KUKA KRL program: MyProgram_050().src

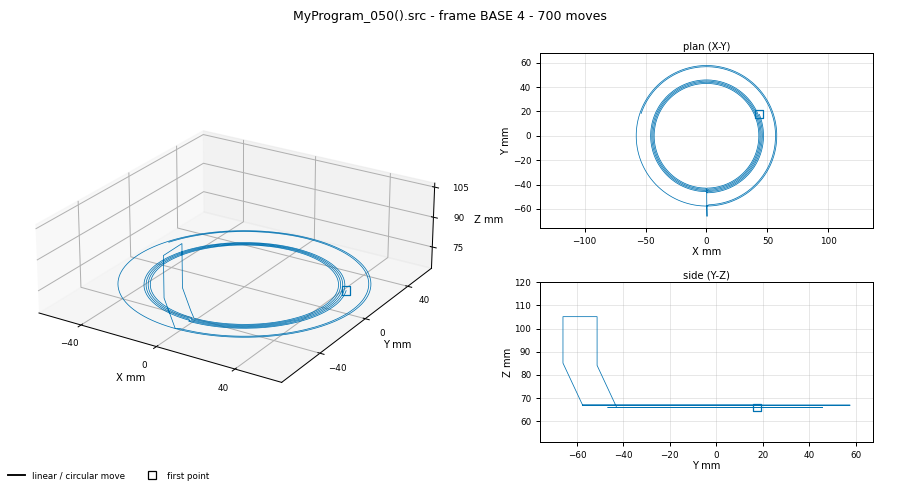
[picture p0: tool path of MyProgram_050().src in frame BASE 4, 700 of 700 moves have a stored position in this frame; points joined in program order, loops and branches not executed]
&ACCESS RVP
&REL 1
&PARAM TEMPLATE = C:\KRC\Roboter\Template\vorgabe
&PARAM EDITMASK = *
DEF MyProgram_050()
; ---- Setting reference (Base) ----
$BASE = BASE_DATA[4]

; --------------------------
; ---- Setting tool (TCP) ----
$TOOL = TOOL_DATA[3]
; --------------------------

$VEL.CP = VEL_APROX_PRINT
Startdeposition()
$VEL.CP = VEL_PRINT
LIN {X 43.3349,Y 17.5684,Z 66,A 14.5783,B 24.8507,C -2.8194,E1 25.1489,E2 68.8422} C_DIS
LIN {X 44.2203,Y 15.2025,Z 66,A 11.1131,B 24.8523,C -2.8036,E1 25.1522,E2 72.3254} C_DIS
LIN {X 45.3904,Y 11.2372,Z 66,A 5.962,B 24.8541,C -2.7869,E1 25.156,E2 77.4863} C_DIS
LIN {X 46.2102,Y 7.1538,Z 66,A 1.4001,B 24.8547,C -2.7815,E1 25.1582,E2 82.0343} C_DIS
LIN {X 46.518,Y 4.7576,Z 66,A -1.6458,B 24.8558,C -2.7707,E1 25.1592,E2 85.0877} C_DIS
LIN {X 46.6896,Y 2.5751,Z 66,A -4.0137,B 24.8561,C -2.7683,E1 25.1596,E2 87.4473} C_DIS
LIN {X 46.7545,Y 0.7633,Z 66,A -6.5593,B 24.8574,C -2.7552,E1 25.1598,E2 90.0088} C_DIS
LIN {X 46.695,Y -2.4713,Z 66,A -10.1755,B 24.858,C -2.7493,E1 25.1595,E2 93.6174} C_DIS
LIN {X 46.5699,Y -4.2183,Z 66,A -12.454,B 24.859,C -2.74,E1 25.1589,E2 95.9043} C_DIS
LIN {X 46.2757,Y -6.7166,Z 66,A -15.3552,B 24.8596,C -2.7338,E1 25.1579,E2 98.8032} C_DIS
LIN {X 45.8823,Y -9.0213,Z 66,A -18.6554,B 24.8614,C -2.7165,E1 25.1562,E2 102.1248} C_DIS
LIN {X 45.206,Y -11.9579,Z 66,A -22.2433,B 24.8624,C -2.7071,E1 25.1538,E2 105.7144} C_DIS
LIN {X 44.3153,Y -14.9224,Z 66,A -25.7557,B 24.863,C -2.7008,E1 25.1508,E2 109.2217} C_DIS
LIN {X 43.3729,Y -17.4745,Z 66,A -29.1739,B 24.8642,C -2.6891,E1 25.1474,E2 112.6486} C_DIS
LIN {X 42.3193,Y -19.8908,Z 66,A -32.2612,B 24.8649,C -2.6822,E1 25.1438,E2 115.7353} C_DIS
LIN {X 40.7412,Y -22.9499,Z 66,A -37.2752,B 24.8676,C -2.6553,E1 25.1371,E2 120.7867} C_DIS
LIN {X 38.8256,Y -26.0596,Z 66,A -41.3629,B 24.8681,C -2.6501,E1 25.1309,E2 124.8663} C_DIS
LIN {X 36.3077,Y -29.4671,Z 66,A -46.4536,B 24.8693,C -2.6384,E1 25.1222,E2 129.9607} C_DIS
LIN {X 34.1441,Y -31.9491,Z 66,A -49.9088,B 24.8693,C -2.6389,E1 25.1158,E2 133.3991} C_DIS
LIN {X 32.775,Y -33.3522,Z 66,A -52.3553,B 24.8699,C -2.6324,E1 25.111,E2 135.8507} C_DIS
LIN {X 31.3542,Y -34.6908,Z 66,A -54.822,B 24.8706,C -2.6255,E1 25.1059,E2 138.3236} C_DIS
LIN {X 29.1349,Y -36.5752,Z 66,A -59.1688,B 24.8727,C -2.6038,E1 25.0964,E2 142.7054} C_DIS
LIN {X 25.3481,Y -39.2942,Z 66,A -63.9176,B 24.8721,C -2.6097,E1 25.0856,E2 147.424} C_DIS
LIN {X 22.2733,Y -41.1151,Z 66,A -69.1086,B 24.8743,C -2.5878,E1 25.0729,E2 152.6516} C_DIS
LIN {X 19.1514,Y -42.6589,Z 66,A -72.7416,B 24.8738,C -2.5922,E1 25.0638,E2 156.2648} C_DIS
LIN {X 16.7047,Y -43.6749,Z 66,A -76.1469,B 24.8745,C -2.585,E1 25.0549,E2 159.6795} C_DIS
LIN {X 14.3201,Y -44.5136,Z 66,A -79.3958,B 24.8752,C -2.5787,E1 25.0463,E2 162.9371} C_DIS
LIN {X 11.2683,Y -45.3827,Z 66,A -82.4317,B 24.8742,C -2.589,E1 25.0382,E2 165.9436} C_DIS
LIN {X 9.0342,Y -45.8799,Z 66,A -86.2122,B 24.876,C -2.5702,E1 25.0277,E2 169.7639} C_DIS
LIN {X 6.7643,Y -46.269,Z 66,A -88.946,B 24.876,C -2.5697,E1 25.0202,E2 172.4964} C_DIS
LIN {X 2.9921,Y -46.665,Z 66,A -93.1614,B 24.8756,C -2.5744,E1 25.0085,E2 176.6981} C_DIS
LIN {X 0.2144,Y -46.7557,Z 66,A -95.0475,B 24.8733,C -2.5983,E1 25.0034,E2 178.5272} C_DIS
Enddeposition()
LIN {X 0.2144,Y -46.7557,Z 66,A -95.0475,B 24.8733,C -2.5983,E1 25.0034,E2 178.5272} C_DIS
Startdeposition()
$VEL.CP = VEL_PRINT
LIN {X 0.8978,Y -45.7928,Z 66,A -94.2069,B 24.8717,C -2.6146,E1 25.0059,E2 177.648} C_DIS
LIN {X 2.9762,Y -45.7048,Z 66,A -91.241,B 24.871,C -2.6216,E1 25.0142,E2 174.6666} C_DIS
LIN {X 6.5228,Y -45.3347,Z 66,A -87.6101,B 24.872,C -2.6106,E1 25.0242,E2 171.0646} C_DIS
LIN {X 7.8991,Y -45.1153,Z 66,A -85.4528,B 24.8712,C -2.6188,E1 25.0301,E2 168.8902} C_DIS
LIN {X 10.8381,Y -44.5008,Z 66,A -81.704,B 24.8709,C -2.6221,E1 25.0404,E2 165.1385} C_DIS
LIN {X 13.368,Y -43.8073,Z 66,A -78.1682,B 24.8701,C -2.63,E1 25.0499,E2 161.5899} C_DIS
LIN {X 15.9038,Y -42.9513,Z 66,A -75.1389,B 24.8702,C -2.6288,E1 25.0578,E2 158.5697} C_DIS
LIN {X 18.2204,Y -42.0213,Z 66,A -72.3421,B 24.8704,C -2.6275,E1 25.065,E2 155.7823} C_DIS
LIN {X 19.5156,Y -41.436,Z 66,A -69.8624,B 24.8689,C -2.6425,E1 25.0714,E2 153.2734} C_DIS
LIN {X 22.8629,Y -39.6867,Z 66,A -65.528,B 24.8688,C -2.6437,E1 25.082,E2 148.9489} C_DIS
LIN {X 24.7649,Y -38.529,Z 66,A -62.1736,B 24.8672,C -2.6591,E1 25.0899,E2 145.5687} C_DIS
LIN {X 28.2935,Y -36.0177,Z 66,A -57.8091,B 24.868,C -2.6512,E1 25.0997,E2 141.2385} C_DIS
LIN {X 30.3014,Y -34.346,Z 66,A -53.7652,B 24.8659,C -2.6725,E1 25.1083,E2 137.16} C_DIS
LIN {X 32.0835,Y -32.6872,Z 66,A -51.4223,B 24.8665,C -2.6667,E1 25.113,E2 134.8403} C_DIS
LIN {X 34.0299,Y -30.6556,Z 66,A -47.0128,B 24.8639,C -2.6918,E1 25.1214,E2 130.3909} C_DIS
LIN {X 35.7191,Y -28.6702,Z 66,A -43.7714,B 24.8631,C -2.6998,E1 25.1271,E2 127.1455} C_DIS
LIN {X 38.0986,Y -25.4232,Z 66,A -39.7855,B 24.8637,C -2.6938,E1 25.1335,E2 123.1933} C_DIS
LIN {X 39.2143,Y -23.6641,Z 66,A -36.3538,B 24.8614,C -2.7165,E1 25.1386,E2 119.7252} C_DIS
LIN {X 41.065,Y -20.2842,Z 66,A -32.2707,B 24.8614,C -2.7165,E1 25.1439,E2 115.6637} C_DIS
LIN {X 41.7032,Y -18.9371,Z 66,A -30.0884,B 24.8602,C -2.728,E1 25.1465,E2 113.466} C_DIS
LIN {X 42.7319,Y -16.4845,Z 66,A -27.0475,B 24.8598,C -2.7326,E1 25.1497,E2 110.4311} C_DIS
LIN {X 43.2185,Y -15.1634,Z 66,A -24.779,B 24.8582,C -2.7475,E1 25.1518,E2 108.1399} C_DIS
LIN {X 44.2475,Y -11.8303,Z 66,A -20.9893,B 24.858,C -2.75,E1 25.1547,E2 104.3659} C_DIS
LIN {X 44.7342,Y -9.8304,Z 66,A -18.011,B 24.8563,C -2.7657,E1 25.1566,E2 101.3678} C_DIS
LIN {X 45.1853,Y -7.488,Z 66,A -14.8477,B 24.855,C -2.7785,E1 25.1581,E2 98.1929} C_DIS
LIN {X 45.6688,Y -3.4865,Z 66,A -10.5749,B 24.8549,C -2.7797,E1 25.1594,E2 93.9426} C_DIS
LIN {X 45.7926,Y -0.9082,Z 66,A -6.6136,B 24.8523,C -2.8038,E1 25.1598,E2 89.9477} C_DIS
LIN {X 45.7713,Y 1.6691,Z 66,A -3.6991,B 24.8519,C -2.808,E1 25.1596,E2 87.0407} C_DIS
LIN {X 45.5857,Y 4.4425,Z 66,A -0.6525,B 24.8516,C -2.8107,E1 25.1589,E2 84.0058} C_DIS
LIN {X 45.3638,Y 6.3188,Z 66,A 1.9954,B 24.8503,C -2.8233,E1 25.1579,E2 81.3435} C_DIS
LIN {X 45.0043,Y 8.508,Z 66,A 4.7588,B 24.8494,C -2.8316,E1 25.1566,E2 78.5769} C_DIS
LIN {X 44.4208,Y 11.161,Z 66,A 7.5921,B 24.8494,C -2.8312,E1 25.1548,E2 75.7609} C_DIS
LIN {X 43.4383,Y 14.5227,Z 66,A 12.5584,B 24.8469,C -2.8551,E1 25.1508,E2 70.7665} C_DIS
LIN {X 42.4975,Y 17.0812,Z 66,A 15.8627,B 24.846,C -2.8628,E1 25.1475,E2 67.4622} C_DIS
LIN {X 41.091,Y 20.2317,Z 66,A 20.3435,B 24.8444,C -2.8778,E1 25.1422,E2 62.9701} C_DIS
LIN {X 39.4422,Y 23.283,Z 66,A 24.8067,B 24.8429,C -2.8915,E1 25.1361,E2 58.4976} C_DIS
LIN {X 37.4354,Y 26.3899,Z 66,A 29.3094,B 24.8419,C -2.9007,E1 25.129,E2 53.9953} C_DIS
LIN {X 35.8889,Y 28.4565,Z 66,A 32.3347,B 24.8415,C -2.9047,E1 25.1239,E2 50.9751} C_DIS
LIN {X 33.9496,Y 30.7449,Z 66,A 35.9504,B 24.8408,C -2.9106,E1 25.1173,E2 47.3616} C_DIS
LIN {X 32.4039,Y 32.37,Z 66,A 38.5786,B 24.8405,C -2.9133,E1 25.1122,E2 44.7381} C_DIS
LIN {X 30.8201,Y 33.8814,Z 66,A 41.5735,B 24.8394,C -2.9233,E1 25.106,E2 41.7318} C_DIS
LIN {X 28.9064,Y 35.5276,Z 66,A 44.755,B 24.8387,C -2.9296,E1 25.0992,E2 38.5476} C_DIS
LIN {X 26.0164,Y 37.6956,Z 66,A 48.8498,B 24.8387,C -2.9299,E1 25.09,E2 34.4667} C_DIS
LIN {X 23.2214,Y 39.4786,Z 66,A 52.9902,B 24.838,C -2.936,E1 25.0802,E2 30.3251} C_DIS
LIN {X 20.8606,Y 40.7752,Z 66,A 56.8481,B 24.8366,C -2.9487,E1 25.0707,E2 26.448} C_DIS
LIN {X 18.7515,Y 41.7872,Z 66,A 60.2609,B 24.8353,C -2.9602,E1 25.0619,E2 23.0165} C_DIS
LIN {X 16.1644,Y 42.8544,Z 66,A 62.9926,B 24.8364,C -2.9507,E1 25.0549,E2 20.3134} C_DIS
LIN {X 13.9943,Y 43.6114,Z 66,A 65.9425,B 24.836,C -2.9542,E1 25.0471,E2 17.3607} C_DIS
LIN {X 11.6913,Y 44.2844,Z 66,A 69.7433,B 24.8343,C -2.9692,E1 25.0368,E2 13.5304} C_DIS
LIN {X 8.6249,Y 44.9822,Z 66,A 73.6023,B 24.8343,C -2.9697,E1 25.0262,E2 9.6749} C_DIS
LIN {X 3.9155,Y 45.634,Z 66,A 78.5134,B 24.836,C -2.9542,E1 25.0127,E2 4.8043} C_DIS
LIN {X 1.0821,Y 45.7888,Z 66,A 82.7236,B 24.8349,C -2.9643,E1 25.0009,E2 0.5713} C_DIS
LIN {X -1.5721,Y 45.7747,Z 66,A 85.9582,B 24.8351,C -2.9621,E1 24.9919,E2 -2.6583} C_DIS
LIN {X -4.9742,Y 45.5306,Z 66,A 90.0108,B 24.8357,C -2.9568,E1 24.9806,E2 -6.7003} C_DIS
LIN {X -7.4603,Y 45.19,Z 66,A 93.4271,B 24.8355,C -2.9589,E1 24.9712,E2 -10.1245} C_DIS
LIN {X -9.7479,Y 44.7522,Z 66,A 96.3601,B 24.8357,C -2.9567,E1 24.9632,E2 -13.056} C_DIS
LIN {X -13.1885,Y 43.8617,Z 66,A 100.5053,B 24.8367,C -2.9478,E1 24.9521,E2 -17.1862} C_DIS
LIN {X -16.3693,Y 42.7765,Z 66,A 104.5263,B 24.8376,C -2.94,E1 24.9415,E2 -21.1966} C_DIS
LIN {X -18.0147,Y 42.1101,Z 66,A 106.8564,B 24.8377,C -2.9384,E1 24.9355,E2 -23.5283} C_DIS
LIN {X -20.0814,Y 41.1647,Z 66,A 109.6892,B 24.8382,C -2.934,E1 24.9284,E2 -26.3577} C_DIS
LIN {X -22.1767,Y 40.075,Z 66,A 113.1651,B 24.838,C -2.9364,E1 24.9198,E2 -29.849} C_DIS
LIN {X -24.6187,Y 38.6228,Z 66,A 116.1352,B 24.8396,C -2.9218,E1 24.9128,E2 -32.7938} C_DIS
LIN {X -26.8632,Y 37.097,Z 66,A 120.1797,B 24.8393,C -2.9241,E1 24.9035,E2 -36.8574} C_DIS
LIN {X -29.4193,Y 35.1045,Z 66,A 123.6418,B 24.8412,C -2.9075,E1 24.896,E2 -40.2928} C_DIS
LIN {X -30.6738,Y 34.0124,Z 66,A 126.2288,B 24.8409,C -2.9096,E1 24.8906,E2 -42.8952} C_DIS
LIN {X -33.081,Y 31.6774,Z 66,A 130.4532,B 24.842,C -2.9,E1 24.8823,E2 -47.1148} C_DIS
LIN {X -35.5132,Y 28.9239,Z 66,A 134.4029,B 24.8442,C -2.8801,E1 24.8752,E2 -51.0347} C_DIS
LIN {X -36.3677,Y 27.8421,Z 66,A 136.3444,B 24.8443,C -2.8784,E1 24.8719,E2 -52.9813} C_DIS
LIN {X -37.8873,Y 25.736,Z 66,A 140.0753,B 24.8446,C -2.8759,E1 24.8659,E2 -56.7246} C_DIS
LIN {X -39.2931,Y 23.5348,Z 66,A 143.5261,B 24.8453,C -2.8692,E1 24.8609,E2 -60.1771} C_DIS
LIN {X -41.2526,Y 19.9,Z 66,A 148.3302,B 24.8474,C -2.8497,E1 24.8547,E2 -64.9601} C_DIS
LIN {X -42.3378,Y 17.4725,Z 66,A 151.8219,B 24.8483,C -2.8419,E1 24.8509,E2 -68.4526} C_DIS
LIN {X -43.324,Y 14.8597,Z 66,A 155.0988,B 24.8497,C -2.8286,E1 24.8478,E2 -71.7163} C_DIS
LIN {X -43.9589,Y 12.861,Z 66,A 157.5559,B 24.8508,C -2.8185,E1 24.8458,E2 -74.1634} C_DIS
LIN {X -44.6534,Y 10.1894,Z 66,A 161.8476,B 24.8508,C -2.8184,E1 24.843,E2 -78.4799} C_DIS
LIN {X -45.4195,Y 5.9038,Z 66,A 166.3561,B 24.8538,C -2.7895,E1 24.841,E2 -82.9462} C_DIS
LIN {X -45.626,Y 4.0058,Z 66,A 169.1778,B 24.8541,C -2.7874,E1 24.8402,E2 -85.7797} C_DIS
LIN {X -45.7994,Y 0.4243,Z 66,A 173.4393,B 24.8558,C -2.7705,E1 24.8398,E2 -90.0265} C_DIS
LIN {X -45.7787,Y -1.4489,Z 66,A 175.8008,B 24.8566,C -2.7634,E1 24.8399,E2 -92.3852} C_DIS
LIN {X -45.6799,Y -3.3462,Z 66,A 178.4462,B 24.857,C -2.7594,E1 24.8404,E2 -95.0368} C_DIS
LIN {X -45.4231,Y -5.876,Z 66,A -178.301,B 24.8579,C -2.7504,E1 24.8414,E2 -98.2877} C_DIS
LIN {X -44.9989,Y -8.5369,Z 66,A -174.9998,B 24.8591,C -2.7393,E1 24.843,E2 -101.5818} C_DIS
LIN {X -44.5654,Y -10.5695,Z 66,A -172.5411,B 24.8601,C -2.7296,E1 24.8445,E2 -104.0319} C_DIS
LIN {X -44.1168,Y -12.3085,Z 66,A -170.3247,B 24.8608,C -2.7226,E1 24.8461,E2 -106.2443} C_DIS
LIN {X -43.5231,Y -14.2665,Z 66,A -167.5795,B 24.8613,C -2.7175,E1 24.8484,E2 -108.9929} C_DIS
LIN {X -42.7238,Y -16.5061,Z 66,A -164.4177,B 24.8619,C -2.7113,E1 24.8515,E2 -112.158} C_DIS
LIN {X -41.6977,Y -18.9494,Z 66,A -161.1109,B 24.8629,C -2.702,E1 24.8552,E2 -115.4607} C_DIS
LIN {X -40.6101,Y -21.1802,Z 66,A -158.1474,B 24.8639,C -2.6918,E1 24.8589,E2 -118.4156} C_DIS
LIN {X -39.2997,Y -23.5238,Z 66,A -154.0372,B 24.8639,C -2.6929,E1 24.8648,E2 -122.5499} C_DIS
LIN {X -37.5087,Y -26.2851,Z 66,A -150.3373,B 24.8654,C -2.6772,E1 24.8705,E2 -126.2305} C_DIS
LIN {X -36.0748,Y -28.2213,Z 66,A -147.7338,B 24.8667,C -2.6645,E1 24.8749,E2 -128.8163} C_DIS
LIN {X -34.2802,Y -30.3759,Z 66,A -144.2149,B 24.8675,C -2.6568,E1 24.8813,E2 -132.3327} C_DIS
LIN {X -32.836,Y -31.9315,Z 66,A -140.544,B 24.8666,C -2.6651,E1 24.8885,E2 -136.0394} C_DIS
LIN {X -30.3871,Y -34.2702,Z 66,A -137.229,B 24.8687,C -2.644,E1 24.8952,E2 -139.3174} C_DIS
LIN {X -28.3039,Y -36.0095,Z 66,A -134.0664,B 24.8697,C -2.6346,E1 24.902,E2 -142.4695} C_DIS
LIN {X -26.0354,Y -37.6823,Z 66,A -130.4029,B 24.8701,C -2.6307,E1 24.9103,E2 -146.1365} C_DIS
LIN {X -24.2685,Y -38.8436,Z 66,A -126.7325,B 24.869,C -2.6415,E1 24.919,E2 -149.8444} C_DIS
LIN {X -21.5446,Y -40.4186,Z 66,A -122.985,B 24.8698,C -2.6336,E1 24.9282,E2 -153.5836} C_DIS
LIN {X -18.9449,Y -41.7,Z 66,A -120.1611,B 24.8713,C -2.6176,E1 24.9353,E2 -156.3767} C_DIS
LIN {X -16.0834,Y -42.885,Z 66,A -116.5309,B 24.8721,C -2.6102,E1 24.9446,E2 -159.9973} C_DIS
LIN {X -14.6878,Y -43.3827,Z 66,A -113.3715,B 24.8703,C -2.6285,E1 24.9531,E2 -163.2062} C_DIS
LIN {X -11.5992,Y -44.3086,Z 66,A -109.5438,B 24.8708,C -2.6228,E1 24.9634,E2 -167.0263} C_DIS
LIN {X -7.817,Y -45.1302,Z 66,A -105.4156,B 24.8721,C -2.6098,E1 24.9746,E2 -171.1283} C_DIS
LIN {X -6.1382,Y -45.3887,Z 66,A -102.6975,B 24.8712,C -2.6187,E1 24.9822,E2 -173.8696} C_DIS
LIN {X -2.2898,Y -45.7446,Z 66,A -97.7991,B 24.8712,C -2.6198,E1 24.9959,E2 -178.7724} C_DIS
LIN {X 0.2079,Y -45.7974,Z 66,A -95.7806,B 24.8728,C -2.6027,E1 25.0014,E2 -180.7503} C_DIS
Enddeposition()
LIN {X 0.2079,Y -45.7974,Z 66,A -95.7806,B 24.8728,C -2.6027,E1 25.0014,E2 -180.7503} C_DIS
Startdeposition()
$VEL.CP = VEL_PRINT
LIN {X -1.0961,Y -44.8291,Z 66,A -98.3264,B 24.8726,C -2.6053,E1 24.9943,E2 -178.2105} C_DIS
LIN {X -3.5551,Y -44.7013,Z 66,A -101.8341,B 24.8731,C -2.5998,E1 24.9845,E2 -174.6884} C_DIS
LIN {X -6.5718,Y -44.3589,Z 66,A -105.07,B 24.8721,C -2.61,E1 24.9756,E2 -171.4747} C_DIS
LIN {X -8.9935,Y -43.9314,Z 66,A -108.9252,B 24.873,C -2.6007,E1 24.9649,E2 -167.593} C_DIS
LIN {X -12.0574,Y -43.1911,Z 66,A -112.9482,B 24.8728,C -2.6031,E1 24.9541,E2 -163.5697} C_DIS
LIN {X -14.9046,Y -42.2931,Z 66,A -116.0557,B 24.8715,C -2.6161,E1 24.9459,E2 -160.4876} C_DIS
LIN {X -17.0497,Y -41.4746,Z 66,A -119.0014,B 24.8712,C -2.6187,E1 24.9382,E2 -157.5417} C_DIS
LIN {X -18.4124,Y -40.8881,Z 66,A -121.5238,B 24.8719,C -2.6119,E1 24.9318,E2 -154.9971} C_DIS
LIN {X -21.075,Y -39.582,Z 66,A -124.5809,B 24.8705,C -2.6267,E1 24.9242,E2 -151.967} C_DIS
LIN {X -22.7553,Y -38.64,Z 66,A -127.5913,B 24.8709,C -2.6225,E1 24.9169,E2 -148.9377} C_DIS
LIN {X -25.0178,Y -37.2153,Z 66,A -130.7665,B 24.87,C -2.631,E1 24.9095,E2 -145.7724} C_DIS
LIN {X -27.1019,Y -35.7265,Z 66,A -133.849,B 24.8692,C -2.639,E1 24.9025,E2 -142.6982} C_DIS
LIN {X -28.5618,Y -34.5698,Z 66,A -136.5508,B 24.8692,C -2.639,E1 24.8966,E2 -139.9863} C_DIS
LIN {X -30.3627,Y -32.9994,Z 66,A -139.6861,B 24.8688,C -2.6438,E1 24.8901,E2 -136.85} C_DIS
LIN {X -32.1877,Y -31.2222,Z 66,A -143.0148,B 24.8682,C -2.6496,E1 24.8835,E2 -133.5209} C_DIS
LIN {X -33.9767,Y -29.2659,Z 66,A -146.3785,B 24.8674,C -2.6573,E1 24.8773,E2 -130.1606} C_DIS
LIN {X -36.0939,Y -26.6098,Z 66,A -150.8068,B 24.8665,C -2.6664,E1 24.8697,E2 -125.733} C_DIS
LIN {X -37.3717,Y -24.7835,Z 66,A -153.7041,B 24.8658,C -2.6728,E1 24.8652,E2 -122.8367} C_DIS
LIN {X -38.9514,Y -22.217,Z 66,A -157.2286,B 24.8644,C -2.6868,E1 24.8602,E2 -119.3275} C_DIS
LIN {X -40.114,Y -20.0422,Z 66,A -161.0936,B 24.8644,C -2.6866,E1 24.8552,E2 -115.4411} C_DIS
LIN {X -41.7879,Y -16.2669,Z 66,A -166.2738,B 24.8628,C -2.7026,E1 24.8496,E2 -110.2705} C_DIS
LIN {X -42.8064,Y -13.359,Z 66,A -169.9902,B 24.8614,C -2.7167,E1 24.8464,E2 -106.5666} C_DIS
LIN {X -43.5529,Y -10.6762,Z 66,A -173.4369,B 24.8602,C -2.7286,E1 24.8439,E2 -103.1284} C_DIS
LIN {X -44.2519,Y -7.2553,Z 66,A -177.8985,B 24.8588,C -2.7422,E1 24.8416,E2 -98.6729} C_DIS
LIN {X -44.5736,Y -4.9035,Z 66,A 178.9456,B 24.858,C -2.7501,E1 24.8405,E2 -95.517} C_DIS
LIN {X -44.7754,Y -2.4523,Z 66,A 175.8262,B 24.8569,C -2.7601,E1 24.8399,E2 -92.4029} C_DIS
LIN {X -44.8382,Y 0.633,Z 66,A 171.627,B 24.8559,C -2.7695,E1 24.8399,E2 -88.2008} C_DIS
LIN {X -44.709,Y 3.4581,Z 66,A 168.237,B 24.8545,C -2.7835,E1 24.8404,E2 -84.8239} C_DIS
LIN {X -44.4713,Y 5.758,Z 66,A 165.5994,B 24.8531,C -2.7965,E1 24.8412,E2 -82.2015} C_DIS
LIN {X -44.1727,Y 7.7235,Z 66,A 162.9182,B 24.8524,C -2.8028,E1 24.8424,E2 -79.5194} C_DIS
LIN {X -43.8881,Y 9.2,Z 66,A 160.6823,B 24.8522,C -2.805,E1 24.8437,E2 -77.2758} C_DIS
LIN {X -43.2527,Y 11.835,Z 66,A 157.2623,B 24.851,C -2.8162,E1 24.846,E2 -73.8626} C_DIS
LIN {X -42.1241,Y 15.3757,Z 66,A 152.4645,B 24.8495,C -2.8301,E1 24.8503,E2 -69.0705} C_DIS
LIN {X -41.1669,Y 17.7808,Z 66,A 149.085,B 24.8486,C -2.8391,E1 24.8539,E2 -65.6938} C_DIS
LIN {X -40.1812,Y 19.9078,Z 66,A 145.9801,B 24.8478,C -2.8465,E1 24.8576,E2 -62.5898} C_DIS
LIN {X -38.9204,Y 22.2723,Z 66,A 142.9464,B 24.8462,C -2.8609,E1 24.8617,E2 -59.5746} C_DIS
LIN {X -38.1209,Y 23.6151,Z 66,A 140.2659,B 24.8465,C -2.8582,E1 24.8656,E2 -56.8739} C_DIS
LIN {X -35.8116,Y 26.9887,Z 66,A 135.1703,B 24.8448,C -2.8737,E1 24.8739,E2 -51.7904} C_DIS
LIN {X -33.5563,Y 29.7456,Z 66,A 130.5424,B 24.8437,C -2.8842,E1 24.8822,E2 -47.1666} C_DIS
LIN {X -30.8479,Y 32.545,Z 66,A 124.9731,B 24.8432,C -2.8886,E1 24.8933,E2 -41.5843} C_DIS
LIN {X -27.7477,Y 35.2265,Z 66,A 120.3765,B 24.8411,C -2.9079,E1 24.9031,E2 -37.0163} C_DIS
LIN {X -25.3402,Y 36.9963,Z 66,A 116.6556,B 24.8401,C -2.9167,E1 24.9116,E2 -33.3036} C_DIS
LIN {X -23.1472,Y 38.4069,Z 66,A 113.4126,B 24.8393,C -2.9239,E1 24.9193,E2 -30.0676} C_DIS
LIN {X -21.121,Y 39.5577,Z 66,A 110.3269,B 24.839,C -2.9275,E1 24.9268,E2 -26.9816} C_DIS
LIN {X -18.8628,Y 40.6823,Z 66,A 107.3467,B 24.838,C -2.9357,E1 24.9343,E2 -24.0133} C_DIS
LIN {X -16.8522,Y 41.5555,Z 66,A 104.3659,B 24.8379,C -2.9372,E1 24.9419,E2 -21.0292} C_DIS
LIN {X -14.3528,Y 42.4835,Z 66,A 100.9401,B 24.8374,C -2.9411,E1 24.9509,E2 -17.606} C_DIS
LIN {X -11.067,Y 43.4555,Z 66,A 95.9669,B 24.8379,C -2.9374,E1 24.9644,E2 -12.6162} C_DIS
LIN {X -7.7207,Y 44.1732,Z 66,A 92.1439,B 24.8366,C -2.9486,E1 24.9748,E2 -8.8155} C_DIS
LIN {X -5.253,Y 44.5337,Z 66,A 89.381,B 24.8357,C -2.9566,E1 24.9824,E2 -6.0697} C_DIS
LIN {X -3.4665,Y 44.7083,Z 66,A 86.7567,B 24.8361,C -2.9529,E1 24.9897,E2 -3.4352} C_DIS
LIN {X -1.4616,Y 44.8187,Z 66,A 84.2173,B 24.836,C -2.9541,E1 24.9968,E2 -0.8982} C_DIS
LIN {X 1.2189,Y 44.826,Z 66,A 80.6447,B 24.8362,C -2.9525,E1 25.0068,E2 2.6779} C_DIS
LIN {X 3.645,Y 44.6942,Z 66,A 77.5581,B 24.8362,C -2.9527,E1 25.0154,E2 5.7626} C_DIS
LIN {X 7.9201,Y 44.1375,Z 66,A 72.0706,B 24.8362,C -2.9517,E1 25.0305,E2 11.2478} C_DIS
LIN {X 10.8981,Y 43.498,Z 66,A 68.0977,B 24.8366,C -2.9484,E1 25.0413,E2 15.2229} C_DIS
LIN {X 13.2841,Y 42.8297,Z 66,A 65.0431,B 24.8366,C -2.948,E1 25.0495,E2 18.2734} C_DIS
LIN {X 15.1067,Y 42.2215,Z 66,A 62.8734,B 24.8364,C -2.9504,E1 25.0552,E2 20.433} C_DIS
LIN {X 16.8697,Y 41.5483,Z 66,A 59.9507,B 24.8376,C -2.9399,E1 25.0629,E2 23.3741} C_DIS
LIN {X 18.7846,Y 40.7183,Z 66,A 56.8402,B 24.8387,C -2.9298,E1 25.0708,E2 26.5006} C_DIS
LIN {X 21.983,Y 39.0848,Z 66,A 52.8769,B 24.8382,C -2.9339,E1 25.0805,E2 30.443} C_DIS
LIN {X 24.6115,Y 37.4851,Z 66,A 49.2337,B 24.8384,C -2.9328,E1 25.0891,E2 34.0772} C_DIS
LIN {X 26.584,Y 36.1125,Z 66,A 46.0376,B 24.8392,C -2.9256,E1 25.0964,E2 37.2791} C_DIS
LIN {X 28.2258,Y 34.8448,Z 66,A 43.2466,B 24.8399,C -2.9185,E1 25.1025,E2 40.0767} C_DIS
LIN {X 30.617,Y 32.7639,Z 66,A 39.5349,B 24.8402,C -2.9164,E1 25.1102,E2 43.7786} C_DIS
LIN {X 32.2368,Y 31.1712,Z 66,A 36.2902,B 24.8415,C -2.9045,E1 25.1166,E2 47.0377} C_DIS
LIN {X 34.044,Y 29.187,Z 66,A 32.8792,B 24.8423,C -2.8972,E1 25.123,E2 50.4507} C_DIS
LIN {X 35.8179,Y 26.9802,Z 66,A 28.6387,B 24.8444,C -2.8779,E1 25.1302,E2 54.7168} C_DIS
LIN {X 37.8808,Y 23.9987,Z 66,A 24.8584,B 24.844,C -2.8812,E1 25.136,E2 58.4707} C_DIS
LIN {X 39.6014,Y 21.0382,Z 66,A 20.3653,B 24.8455,C -2.8676,E1 25.1422,E2 62.9726} C_DIS
LIN {X 40.88,Y 18.4303,Z 66,A 16.6973,B 24.8465,C -2.8582,E1 25.1466,E2 66.6431} C_DIS
LIN {X 41.7901,Y 16.2621,Z 66,A 13.7995,B 24.8472,C -2.8516,E1 25.1496,E2 69.5406} C_DIS
LIN {X 42.5408,Y 14.1828,Z 66,A 11.3118,B 24.8475,C -2.8494,E1 25.1519,E2 72.0193} C_DIS
LIN {X 43.3076,Y 11.6321,Z 66,A 7.8263,B 24.8487,C -2.8379,E1 25.1547,E2 75.5122} C_DIS
LIN {X 44.0583,Y 8.3494,Z 66,A 2.2922,B 24.8524,C -2.8027,E1 25.1578,E2 81.0974} C_DIS
LIN {X 44.7147,Y 3.3861,Z 66,A -3.5085,B 24.8534,C -2.7936,E1 25.1595,E2 86.8852} C_DIS
LIN {X 44.8366,Y 0.7345,Z 66,A -6.9497,B 24.8546,C -2.7821,E1 25.1598,E2 90.3332} C_DIS
LIN {X 44.7679,Y -2.5887,Z 66,A -10.6733,B 24.855,C -2.7782,E1 25.1594,E2 94.0437} C_DIS
LIN {X 44.6107,Y -4.555,Z 66,A -13.3542,B 24.8562,C -2.7674,E1 25.1587,E2 96.7345} C_DIS
LIN {X 44.2502,Y -7.2652,Z 66,A -16.9407,B 24.8575,C -2.7547,E1 25.1572,E2 100.3299} C_DIS
LIN {X 43.7101,Y -10.0141,Z 66,A -20.2533,B 24.8581,C -2.7484,E1 25.1552,E2 103.638} C_DIS
LIN {X 43.2886,Y -11.7027,Z 66,A -22.4468,B 24.8588,C -2.7421,E1 25.1537,E2 105.8339} C_DIS
LIN {X 42.6153,Y -13.9565,Z 66,A -25.155,B 24.8592,C -2.7383,E1 25.1514,E2 108.5357} C_DIS
LIN {X 42.0653,Y -15.5358,Z 66,A -27.6257,B 24.8605,C -2.7257,E1 25.1491,E2 111.0222} C_DIS
LIN {X 40.9748,Y -18.2179,Z 66,A -31.0418,B 24.8611,C -2.7199,E1 25.1454,E2 114.4335} C_DIS
LIN {X 40.3276,Y -19.6102,Z 66,A -32.9184,B 24.8615,C -2.7156,E1 25.1431,E2 116.31} C_DIS
LIN {X 39.658,Y -20.9299,Z 66,A -35.3352,B 24.863,C -2.7007,E1 25.1399,E2 118.7493} C_DIS
LIN {X 37.6383,Y -24.3771,Z 66,A -40.0826,B 24.8638,C -2.6928,E1 25.1331,E2 123.4912} C_DIS
LIN {X 36.7657,Y -25.6737,Z 66,A -42.9474,B 24.8659,C -2.672,E1 25.1284,E2 126.3913} C_DIS
LIN {X 34.7631,Y -28.3265,Z 66,A -46.8016,B 24.8663,C -2.6679,E1 25.1217,E2 130.2372} C_DIS
LIN {X 31.9301,Y -31.4853,Z 66,A -51.7504,B 24.8668,C -2.6629,E1 25.1123,E2 135.1761} C_DIS
LIN {X 29.5991,Y -33.6862,Z 66,A -56.1817,B 24.8684,C -2.6477,E1 25.1031,E2 139.6256} C_DIS
LIN {X 27.6126,Y -35.3334,Z 66,A -59.1822,B 24.8686,C -2.6458,E1 25.0966,E2 142.6194} C_DIS
LIN {X 25.181,Y -37.1049,Z 66,A -62.3135,B 24.8681,C -2.6503,E1 25.0896,E2 145.7289} C_DIS
LIN {X 23.1172,Y -38.4251,Z 66,A -65.7492,B 24.8692,C -2.6392,E1 25.0814,E2 149.1798} C_DIS
LIN {X 21.2211,Y -39.5037,Z 66,A -68.8802,B 24.8703,C -2.6286,E1 25.0737,E2 152.3269} C_DIS
LIN {X 18.8244,Y -40.7001,Z 66,A -72.2364,B 24.8707,C -2.6244,E1 25.0653,E2 155.6843} C_DIS
LIN {X 16.3931,Y -41.7387,Z 66,A -75.6012,B 24.8711,C -2.6199,E1 25.0566,E2 159.0522} C_DIS
LIN {X 13.728,Y -42.6896,Z 66,A -79.0747,B 24.8713,C -2.6177,E1 25.0474,E2 162.5239} C_DIS
LIN {X 11.424,Y -43.363,Z 66,A -82.1135,B 24.8716,C -2.6149,E1 25.0392,E2 165.5643} C_DIS
LIN {X 9.383,Y -43.8498,Z 66,A -84.6722,B 24.8716,C -2.6144,E1 25.0323,E2 168.1207} C_DIS
LIN {X 7.4549,Y -44.2185,Z 66,A -87.3757,B 24.8722,C -2.6094,E1 25.0248,E2 170.8333} C_DIS
LIN {X 4.8255,Y -44.5821,Z 66,A -90.8358,B 24.8725,C -2.6062,E1 25.0152,E2 174.2983} C_DIS
LIN {X 2.2365,Y -44.787,Z 66,A -94.4946,B 24.8731,C -2.5995,E1 25.005,E2 177.9714} C_DIS
LIN {X 0.2157,Y -44.8397,Z 66,A -96.6399,B 24.8725,C -2.6056,E1 24.999,E2 180.102} C_DIS
Enddeposition()
LIN {X 0.2157,Y -44.8397,Z 66,A -96.6399,B 24.8725,C -2.6056,E1 24.999,E2 180.102} C_DIS
Startdeposition()
$VEL.CP = VEL_PRINT
LIN {X 1.8251,Y -43.8455,Z 66,A -93.5919,B 24.8694,C -2.6374,E1 25.0077,E2 176.9788} C_DIS
LIN {X 3.5917,Y -43.7363,Z 66,A -90.8078,B 24.8686,C -2.6458,E1 25.0155,E2 174.1761} C_DIS
LIN {X 5.9074,Y -43.4844,Z 66,A -87.7302,B 24.8683,C -2.6483,E1 25.0241,E2 171.0951} C_DIS
LIN {X 9.227,Y -42.9021,Z 66,A -83.256,B 24.8678,C -2.653,E1 25.0364,E2 166.6148} C_DIS
LIN {X 11.7602,Y -42.2783,Z 66,A -79.8983,B 24.8676,C -2.6557,E1 25.0454,E2 163.2559} C_DIS
LIN {X 14.0845,Y -41.5619,Z 66,A -76.7299,B 24.8672,C -2.6593,E1 25.0539,E2 160.0848} C_DIS
LIN {X 17.4642,Y -40.2587,Z 66,A -72.6227,B 24.8676,C -2.6555,E1 25.0645,E2 155.9958} C_DIS
LIN {X 20.0165,Y -39.0526,Z 66,A -67.9865,B 24.8654,C -2.6773,E1 25.0762,E2 151.3203} C_DIS
LIN {X 22.2262,Y -37.8387,Z 66,A -65.2327,B 24.8657,C -2.6739,E1 25.0828,E2 148.5828} C_DIS
LIN {X 24.1935,Y -36.6119,Z 66,A -62.2631,B 24.8653,C -2.6787,E1 25.0898,E2 145.6115} C_DIS
LIN {X 25.5963,Y -35.6455,Z 66,A -59.6142,B 24.8641,C -2.6904,E1 25.0959,E2 142.944} C_DIS
LIN {X 27.7223,Y -34.0183,Z 66,A -56.0161,B 24.8631,C -2.6997,E1 25.1038,E2 139.3374} C_DIS
LIN {X 29.8614,Y -32.1575,Z 66,A -52.6839,B 24.8629,C -2.7016,E1 25.1106,E2 136.0141} C_DIS
LIN {X 31.6738,Y -30.3733,Z 66,A -49.3955,B 24.8622,C -2.709,E1 25.1171,E2 132.7222} C_DIS
LIN {X 34.0551,Y -27.6769,Z 66,A -45.124,B 24.8617,C -2.7133,E1 25.1249,E2 128.4598} C_DIS
LIN {X 35.4035,Y -25.9297,Z 66,A -42.3037,B 24.8611,C -2.7198,E1 25.1297,E2 125.6375} C_DIS
LIN {X 36.3735,Y -24.5504,Z 66,A -39.756,B 24.8598,C -2.732,E1 25.1337,E2 123.0735} C_DIS
LIN {X 37.9884,Y -21.9691,Z 66,A -35.2804,B 24.8577,C -2.7522,E1 25.1402,E2 118.573} C_DIS
LIN {X 39.6286,Y -18.8505,Z 66,A -31.1702,B 24.8573,C -2.7566,E1 25.1453,E2 114.4742} C_DIS
LIN {X 40.736,Y -16.319,Z 66,A -27.7709,B 24.8565,C -2.7636,E1 25.149,E2 111.0771} C_DIS
LIN {X 41.5493,Y -14.1212,Z 66,A -24.3977,B 24.855,C -2.7786,E1 25.1522,E2 107.6874} C_DIS
LIN {X 42.3295,Y -11.575,Z 66,A -21.3071,B 24.8546,C -2.7822,E1 25.1546,E2 104.6058} C_DIS
LIN {X 42.853,Y -9.4548,Z 66,A -18.2142,B 24.8532,C -2.7955,E1 25.1565,E2 101.4994} C_DIS
LIN {X 43.3151,Y -7.0425,Z 66,A -14.9587,B 24.852,C -2.8064,E1 25.1581,E2 98.2372} C_DIS
LIN {X 43.6295,Y -4.7149,Z 66,A -12.0901,B 24.8514,C -2.8124,E1 25.1591,E2 95.3713} C_DIS
LIN {X 43.807,Y -2.5945,Z 66,A -9.3751,B 24.8506,C -2.82,E1 25.1596,E2 92.6544} C_DIS
LIN {X 43.8812,Y -0.4433,Z 66,A -6.4724,B 24.8495,C -2.8305,E1 25.1598,E2 89.7441} C_DIS
LIN {X 43.8088,Y 2.5627,Z 66,A -2.0793,B 24.8472,C -2.8514,E1 25.1592,E2 85.3278} C_DIS
LIN {X 43.5582,Y 5.3344,Z 66,A 1.0167,B 24.8471,C -2.8528,E1 25.1583,E2 82.2468} C_DIS
LIN {X 43.1773,Y 7.841,Z 66,A 5.3551,B 24.844,C -2.8818,E1 25.1562,E2 77.8652} C_DIS
LIN {X 42.2856,Y 11.7336,Z 66,A 9.4473,B 24.8445,C -2.8769,E1 25.1534,E2 73.8083} C_DIS
LIN {X 41.7179,Y 13.6156,Z 66,A 12.1006,B 24.8435,C -2.8859,E1 25.1511,E2 71.1486} C_DIS
LIN {X 40.808,Y 16.1391,Z 66,A 15.525,B 24.8426,C -2.8946,E1 25.1478,E2 67.7229} C_DIS
LIN {X 39.7955,Y 18.4952,Z 66,A 18.8419,B 24.8416,C -2.9033,E1 25.144,E2 64.4033} C_DIS
LIN {X 38.956,Y 20.2042,Z 66,A 21.4896,B 24.8406,C -2.9129,E1 25.1406,E2 61.7468} C_DIS
LIN {X 37.7993,Y 22.2929,Z 66,A 24.3165,B 24.8402,C -2.9159,E1 25.1367,E2 58.9275} C_DIS
LIN {X 36.6128,Y 24.1922,Z 66,A 27.2273,B 24.8394,C -2.9231,E1 25.1323,E2 56.0143} C_DIS
LIN {X 35.1474,Y 26.276,Z 66,A 30.2972,B 24.839,C -2.9267,E1 25.1273,E2 52.9508} C_DIS
LIN {X 33.9943,Y 27.7519,Z 66,A 33.0742,B 24.8378,C -2.9381,E1 25.1224,E2 50.1596} C_DIS
LIN {X 32.402,Y 29.5952,Z 66,A 36.3758,B 24.8368,C -2.9473,E1 25.1163,E2 46.8511} C_DIS
LIN {X 30.6006,Y 31.4548,Z 66,A 39.6157,B 24.8362,C -2.9519,E1 25.1099,E2 43.614} C_DIS
LIN {X 28.7215,Y 33.1793,Z 66,A 42.9458,B 24.8355,C -2.9583,E1 25.1029,E2 40.2819} C_DIS
LIN {X 26.3865,Y 35.0644,Z 66,A 46.8908,B 24.8347,C -2.9657,E1 25.0943,E2 36.3339} C_DIS
LIN {X 24.6389,Y 36.3136,Z 66,A 49.2448,B 24.835,C -2.9628,E1 25.0889,E2 33.9949} C_DIS
LIN {X 22.9799,Y 37.3861,Z 66,A 52.0533,B 24.8342,C -2.9705,E1 25.0823,E2 31.1773} C_DIS
LIN {X 21.1659,Y 38.4424,Z 66,A 54.8527,B 24.8336,C -2.9752,E1 25.0754,E2 28.3749} C_DIS
LIN {X 19.2052,Y 39.458,Z 66,A 57.8202,B 24.8331,C -2.9801,E1 25.068,E2 25.4038} C_DIS
LIN {X 17.1242,Y 40.4043,Z 66,A 61.1792,B 24.832,C -2.9893,E1 25.0594,E2 22.031} C_DIS
LIN {X 14.7005,Y 41.348,Z 66,A 64.0143,B 24.8327,C -2.9835,E1 25.052,E2 19.2158} C_DIS
LIN {X 12.4374,Y 42.0841,Z 66,A 67.3326,B 24.8321,C -2.9891,E1 25.0431,E2 15.8902} C_DIS
LIN {X 10.0991,Y 42.7057,Z 66,A 70.5928,B 24.8317,C -2.9925,E1 25.0343,E2 12.6267} C_DIS
LIN {X 7.3725,Y 43.2599,Z 66,A 74.2584,B 24.8315,C -2.9943,E1 25.0242,E2 8.9608} C_DIS
LIN {X 4.6704,Y 43.6343,Z 66,A 77.6396,B 24.8317,C -2.9923,E1 25.0149,E2 5.5871} C_DIS
LIN {X 2.2041,Y 43.8284,Z 66,A 80.7459,B 24.8319,C -2.9904,E1 25.0062,E2 2.4865} C_DIS
LIN {X -0.0167,Y 43.8842,Z 66,A 83.7763,B 24.8318,C -2.9919,E1 24.9978,E2 -0.5471} C_DIS
LIN {X -3.3038,Y 43.7591,Z 66,A 87.9949,B 24.8321,C -2.9892,E1 24.986,E2 -4.7605} C_DIS
LIN {X -5.6989,Y 43.5119,Z 66,A 91.1172,B 24.8323,C -2.9872,E1 24.9774,E2 -7.88} C_DIS
LIN {X -8.0308,Y 43.1427,Z 66,A 94.3102,B 24.8323,C -2.9865,E1 24.9686,E2 -11.0745} C_DIS
LIN {X -10.5586,Y 42.5945,Z 66,A 98.2857,B 24.8318,C -2.9919,E1 24.9577,E2 -15.0681} C_DIS
LIN {X -14.0144,Y 41.5855,Z 66,A 102.3664,B 24.8333,C -2.978,E1 24.9469,E2 -19.1229} C_DIS
LIN {X -16.5333,Y 40.6498,Z 66,A 105.5013,B 24.8344,C -2.9683,E1 24.9388,E2 -22.2414} C_DIS
LIN {X -18.1393,Y 39.9592,Z 66,A 108.1192,B 24.8343,C -2.9695,E1 24.9321,E2 -24.8685} C_DIS
LIN {X -20.2207,Y 38.9474,Z 66,A 111.2285,B 24.8347,C -2.9659,E1 24.9243,E2 -27.9774} C_DIS
LIN {X -22.497,Y 37.6787,Z 66,A 114.5969,B 24.8354,C -2.9596,E1 24.9162,E2 -31.3406} C_DIS
LIN {X -24.5931,Y 36.3446,Z 66,A 118.0066,B 24.8358,C -2.9556,E1 24.9082,E2 -34.7521} C_DIS
LIN {X -27.5484,Y 34.1593,Z 66,A 122.4415,B 24.8375,C -2.9411,E1 24.8984,E2 -39.1683} C_DIS
LIN {X -29.1596,Y 32.7948,Z 66,A 125.5381,B 24.8376,C -2.9393,E1 24.8919,E2 -42.2727} C_DIS
LIN {X -31.3438,Y 30.714,Z 66,A 129.3096,B 24.8389,C -2.928,E1 24.8844,E2 -46.033} C_DIS
LIN {X -32.669,Y 29.3,Z 66,A 131.9949,B 24.8394,C -2.9238,E1 24.8793,E2 -48.72} C_DIS
LIN {X -34.48,Y 27.1458,Z 66,A 135.3497,B 24.8408,C -2.9104,E1 24.8734,E2 -52.0586} C_DIS
LIN {X -35.699,Y 25.5214,Z 66,A 138.3714,B 24.8411,C -2.908,E1 24.8684,E2 -55.089} C_DIS
LIN {X -37.0707,Y 23.4853,Z 66,A 141.7608,B 24.8418,C -2.9014,E1 24.8633,E2 -58.4798} C_DIS
LIN {X -38.5405,Y 20.9853,Z 66,A 145.4611,B 24.8431,C -2.8897,E1 24.8582,E2 -62.1714} C_DIS
LIN {X -39.675,Y 18.7527,Z 66,A 148.6868,B 24.8442,C -2.8797,E1 24.8542,E2 -65.3905} C_DIS
LIN {X -40.668,Y 16.4887,Z 66,A 151.9134,B 24.8452,C -2.8701,E1 24.8507,E2 -68.6121} C_DIS
LIN {X -41.4999,Y 14.2657,Z 66,A 154.949,B 24.8463,C -2.86,E1 24.8479,E2 -71.6407} C_DIS
LIN {X -42.1707,Y 12.14,Z 66,A 157.5223,B 24.8477,C -2.8471,E1 24.8458,E2 -74.1979} C_DIS
LIN {X -42.6209,Y 10.4502,Z 66,A 160.4103,B 24.8477,C -2.8471,E1 24.8438,E2 -77.1031} C_DIS
LIN {X -43.2328,Y 7.5312,Z 66,A 163.8712,B 24.8496,C -2.8299,E1 24.8419,E2 -80.5431} C_DIS
LIN {X -43.4874,Y 5.8847,Z 66,A 166.4662,B 24.8497,C -2.8281,E1 24.8409,E2 -83.1492} C_DIS
LIN {X -43.7636,Y 3.2485,Z 66,A 169.9016,B 24.8509,C -2.8169,E1 24.8401,E2 -86.5784} C_DIS
LIN {X -43.8754,Y 0.842,Z 66,A 173.083,B 24.8519,C -2.8074,E1 24.8398,E2 -89.7564} C_DIS
LIN {X -43.8483,Y -1.7598,Z 66,A 176.497,B 24.853,C -2.797,E1 24.84,E2 -93.166} C_DIS
LIN {X -43.6843,Y -4.1784,Z 66,A 179.7478,B 24.854,C -2.7882,E1 24.8408,E2 -96.4151} C_DIS
LIN {X -43.3723,Y -6.6782,Z 66,A -176.9762,B 24.855,C -2.7779,E1 24.842,E2 -99.6862} C_DIS
LIN {X -42.8751,Y -9.3531,Z 66,A -173.8791,B 24.8567,C -2.7617,E1 24.8437,E2 -102.7628} C_DIS
LIN {X -42.2911,Y -11.7139,Z 66,A -169.7916,B 24.8566,C -2.7632,E1 24.8466,E2 -106.8777} C_DIS
LIN {X -41.2842,Y -14.8785,Z 66,A -165.84,B 24.8584,C -2.746,E1 24.8502,E2 -110.8105} C_DIS
LIN {X -40.329,Y -17.3014,Z 66,A -162.4858,B 24.8594,C -2.7358,E1 24.8537,E2 -114.1591} C_DIS
LIN {X -39.3435,Y -19.4383,Z 66,A -159.3129,B 24.8602,C -2.7286,E1 24.8575,E2 -117.3321} C_DIS
LIN {X -38.063,Y -21.8396,Z 66,A -155.6909,B 24.861,C -2.7201,E1 24.8624,E2 -120.9527} C_DIS
LIN {X -36.6758,Y -24.0967,Z 66,A -152.5261,B 24.8623,C -2.7077,E1 24.8671,E2 -124.1039} C_DIS
LIN {X -35.5943,Y -25.6678,Z 66,A -149.7317,B 24.8625,C -2.7054,E1 24.8717,E2 -126.9066} C_DIS
LIN {X -34.0224,Y -27.7172,Z 66,A -146.4134,B 24.8634,C -2.6969,E1 24.8774,E2 -130.2201} C_DIS
LIN {X -32.4148,Y -29.5813,Z 66,A -143.1417,B 24.8641,C -2.6906,E1 24.8835,E2 -133.4914} C_DIS
LIN {X -30.6867,Y -31.3707,Z 66,A -139.9179,B 24.8648,C -2.6835,E1 24.8898,E2 -136.7121} C_DIS
LIN {X -28.808,Y -33.1038,Z 66,A -136.2072,B 24.8649,C -2.6821,E1 24.8976,E2 -140.434} C_DIS
LIN {X -26.9346,Y -34.6457,Z 66,A -133.6658,B 24.8663,C -2.6681,E1 24.9031,E2 -142.9514} C_DIS
LIN {X -25.4062,Y -35.7812,Z 66,A -130.9707,B 24.8665,C -2.6667,E1 24.9092,E2 -145.6529} C_DIS
LIN {X -23.3872,Y -37.1325,Z 66,A -127.7843,B 24.8669,C -2.6621,E1 24.9166,E2 -148.8386} C_DIS
LIN {X -21.1889,Y -38.4293,Z 66,A -124.4419,B 24.8674,C -2.6577,E1 24.9247,E2 -152.1803} C_DIS
LIN {X -18.9586,Y -39.5767,Z 66,A -121.1192,B 24.8677,C -2.6545,E1 24.933,E2 -155.5041} C_DIS
LIN {X -16.9063,Y -40.4959,Z 66,A -118.145,B 24.8679,C -2.6519,E1 24.9407,E2 -158.4792} C_DIS
LIN {X -15.0037,Y -41.2389,Z 66,A -115.7312,B 24.8685,C -2.646,E1 24.947,E2 -160.8838} C_DIS
LIN {X -13.2863,Y -41.8238,Z 66,A -113.0218,B 24.8682,C -2.6491,E1 24.9542,E2 -163.6055} C_DIS
LIN {X -11.3765,Y -42.3832,Z 66,A -110.4899,B 24.8685,C -2.6465,E1 24.961,E2 -166.1353} C_DIS
LIN {X -8.2381,Y -43.1033,Z 66,A -106.3235,B 24.8687,C -2.6441,E1 24.9724,E2 -170.301} C_DIS
LIN {X -5.851,Y -43.4919,Z 66,A -103.2395,B 24.8689,C -2.6422,E1 24.9809,E2 -173.3832} C_DIS
LIN {X -3.6327,Y -43.733,Z 66,A -100.1543,B 24.8687,C -2.6446,E1 24.9895,E2 -176.4758} C_DIS
LIN {X 0.2068,Y -43.883,Z 66,A -97.5615,B 24.8722,C -2.6087,E1 24.9965,E2 -178.9838} C_DIS
Enddeposition()
LIN {X 0.2068,Y -43.883,Z 66,A -97.5615,B 24.8722,C -2.6087,E1 24.9965,E2 -178.9838} C_DIS
Startdeposition()
$VEL.CP = VEL_PRINT
LIN {X -0.6748,Y -42.9192,Z 66,A -98.0378,B 24.8695,C -2.6358,E1 24.9953,E2 -178.5718} C_DIS
LIN {X -3.1711,Y -42.8077,Z 66,A -101.2845,B 24.8695,C -2.6369,E1 24.9863,E2 -175.3268} C_DIS
LIN {X -5.3781,Y -42.5864,Z 66,A -104.1512,B 24.8693,C -2.6387,E1 24.9783,E2 -172.4623} C_DIS
LIN {X -7.7318,Y -42.2225,Z 66,A -107.416,B 24.8693,C -2.6384,E1 24.9693,E2 -169.1938} C_DIS
LIN {X -9.9214,Y -41.7622,Z 66,A -110.3965,B 24.8691,C -2.6399,E1 24.9612,E2 -166.213} C_DIS
LIN {X -12.0777,Y -41.1903,Z 66,A -113.2409,B 24.8688,C -2.6436,E1 24.9536,E2 -163.373} C_DIS
LIN {X -13.9666,Y -40.5886,Z 66,A -116.1164,B 24.8688,C -2.6425,E1 24.9459,E2 -160.4896} C_DIS
LIN {X -16.1091,Y -39.787,Z 66,A -118.957,B 24.8683,C -2.6482,E1 24.9385,E2 -157.6564} C_DIS
LIN {X -18.0375,Y -38.9507,Z 66,A -121.8282,B 24.8681,C -2.6503,E1 24.9312,E2 -154.7833} C_DIS
LIN {X -20.0149,Y -37.9725,Z 66,A -124.906,B 24.8679,C -2.6522,E1 24.9236,E2 -151.7017} C_DIS
LIN {X -22.0728,Y -36.815,Z 66,A -127.9543,B 24.8673,C -2.6579,E1 24.9162,E2 -148.6579} C_DIS
LIN {X -23.9481,Y -35.6232,Z 66,A -130.9221,B 24.8669,C -2.6624,E1 24.9093,E2 -145.6911} C_DIS
LIN {X -25.5723,Y -34.4761,Z 66,A -133.6484,B 24.8665,C -2.6659,E1 24.9031,E2 -142.9636} C_DIS
LIN {X -27.4472,Y -33.0024,Z 66,A -136.8912,B 24.866,C -2.6708,E1 24.8961,E2 -139.7205} C_DIS
LIN {X -29.2658,Y -31.4015,Z 66,A -140.2192,B 24.8655,C -2.676,E1 24.8892,E2 -136.3914} C_DIS
LIN {X -31.0893,Y -29.5973,Z 66,A -143.5163,B 24.8647,C -2.6846,E1 24.8827,E2 -133.1009} C_DIS
LIN {X -32.6708,Y -27.841,Z 66,A -146.7566,B 24.8641,C -2.6906,E1 24.8768,E2 -129.8603} C_DIS
LIN {X -34.2257,Y -25.9061,Z 66,A -150.1648,B 24.8634,C -2.6972,E1 24.8709,E2 -126.4517} C_DIS
LIN {X -35.6901,Y -23.8489,Z 66,A -153.5048,B 24.8625,C -2.7058,E1 24.8656,E2 -123.1159} C_DIS
LIN {X -36.8982,Y -21.9326,Z 66,A -156.497,B 24.8617,C -2.714,E1 24.8613,E2 -120.1278} C_DIS
LIN {X -38.0532,Y -19.8609,Z 66,A -159.7375,B 24.8609,C -2.7215,E1 24.857,E2 -116.8882} C_DIS
LIN {X -39.193,Y -17.5046,Z 66,A -163.2619,B 24.8599,C -2.7308,E1 24.8528,E2 -113.3668} C_DIS
LIN {X -40.1872,Y -15.0833,Z 66,A -166.7128,B 24.8589,C -2.7412,E1 24.8493,E2 -109.9214} C_DIS
LIN {X -40.9465,Y -12.8797,Z 66,A -169.9968,B 24.8581,C -2.7483,E1 24.8464,E2 -106.6356} C_DIS
LIN {X -41.6647,Y -10.3233,Z 66,A -173.4727,B 24.857,C -2.7596,E1 24.844,E2 -103.1665} C_DIS
LIN {X -42.2011,Y -7.8485,Z 66,A -176.7157,B 24.8557,C -2.7714,E1 24.8422,E2 -99.9326} C_DIS
LIN {X -42.5348,Y -5.7732,Z 66,A -179.6541,B 24.855,C -2.7785,E1 24.841,E2 -96.9938} C_DIS
LIN {X -42.7745,Y -3.5877,Z 66,A 177.5641,B 24.8539,C -2.7893,E1 24.8402,E2 -94.2211} C_DIS
LIN {X -42.8954,Y -1.5854,Z 66,A 174.6385,B 24.8533,C -2.7949,E1 24.8398,E2 -91.2913} C_DIS
LIN {X -42.9198,Y 0.6371,Z 66,A 171.8712,B 24.852,C -2.8064,E1 24.8398,E2 -88.5349} C_DIS
LIN {X -42.8441,Y 2.6344,Z 66,A 169.0795,B 24.8513,C -2.8134,E1 24.8402,E2 -85.7431} C_DIS
LIN {X -42.6631,Y 4.7297,Z 66,A 166.2993,B 24.8503,C -2.8226,E1 24.841,E2 -82.9681} C_DIS
LIN {X -42.381,Y 6.8133,Z 66,A 163.7687,B 24.8491,C -2.8344,E1 24.842,E2 -80.4507} C_DIS
LIN {X -42.0426,Y 8.656,Z 66,A 160.9656,B 24.8486,C -2.8388,E1 24.8435,E2 -77.6416} C_DIS
LIN {X -41.5297,Y 10.8534,Z 66,A 157.7498,B 24.8478,C -2.8459,E1 24.8456,E2 -74.4238} C_DIS
LIN {X -40.7915,Y 13.3629,Z 66,A 154.2335,B 24.8467,C -2.8563,E1 24.8485,E2 -70.9123} C_DIS
LIN {X -39.898,Y 15.8324,Z 66,A 150.7746,B 24.8455,C -2.8673,E1 24.8519,E2 -67.4603} C_DIS
LIN {X -38.9746,Y 17.9856,Z 66,A 147.7126,B 24.8445,C -2.8773,E1 24.8554,E2 -64.4053} C_DIS
LIN {X -38.0219,Y 19.9206,Z 66,A 144.6476,B 24.8438,C -2.8835,E1 24.8593,E2 -61.3387} C_DIS
LIN {X -36.8041,Y 22.0911,Z 66,A 141.4558,B 24.8426,C -2.8943,E1 24.8637,E2 -58.1561} C_DIS
LIN {X -35.6158,Y 23.959,Z 66,A 138.492,B 24.8417,C -2.9023,E1 24.8682,E2 -55.1965} C_DIS
LIN {X -34.2336,Y 25.8957,Z 66,A 135.1733,B 24.841,C -2.909,E1 24.8737,E2 -51.8779} C_DIS
LIN {X -32.6354,Y 27.8826,Z 66,A 131.7657,B 24.84,C -2.9176,E1 24.8798,E2 -48.4751} C_DIS
LIN {X -31.0659,Y 29.6218,Z 66,A 128.5804,B 24.8393,C -2.9245,E1 24.8858,E2 -45.2923} C_DIS
LIN {X -29.2489,Y 31.4174,Z 66,A 125.215,B 24.8384,C -2.9329,E1 24.8926,E2 -41.9332} C_DIS
LIN {X -27.4344,Y 33.013,Z 66,A 121.9424,B 24.8376,C -2.9394,E1 24.8995,E2 -38.6633} C_DIS
LIN {X -25.5521,Y 34.4912,Z 66,A 118.7453,B 24.8369,C -2.946,E1 24.9066,E2 -35.4702} C_DIS
LIN {X -23.4979,Y 35.9218,Z 66,A 115.4179,B 24.8362,C -2.9525,E1 24.9143,E2 -32.1475} C_DIS
LIN {X -21.6092,Y 37.0891,Z 66,A 112.5079,B 24.8355,C -2.9585,E1 24.9212,E2 -29.2428} C_DIS
LIN {X -19.6615,Y 38.1569,Z 66,A 109.5344,B 24.835,C -2.9632,E1 24.9286,E2 -26.2723} C_DIS
LIN {X -17.512,Y 39.1897,Z 66,A 106.1858,B 24.8347,C -2.9659,E1 24.9371,E2 -22.9218} C_DIS
LIN {X -15.084,Y 40.1869,Z 66,A 102.7233,B 24.8341,C -2.9711,E1 24.946,E2 -19.4641} C_DIS
LIN {X -12.8387,Y 40.9594,Z 66,A 99.6412,B 24.8336,C -2.9759,E1 24.9542,E2 -16.3879} C_DIS
LIN {X -10.8074,Y 41.5417,Z 66,A 96.8959,B 24.8331,C -2.9798,E1 24.9616,E2 -13.6474} C_DIS
LIN {X -8.7621,Y 42.0208,Z 66,A 94.0088,B 24.833,C -2.9811,E1 24.9694,E2 -10.7599} C_DIS
LIN {X -6.4142,Y 42.4427,Z 66,A 90.7392,B 24.8329,C -2.9822,E1 24.9784,E2 -7.4898} C_DIS
LIN {X -4.0555,Y 42.7325,Z 66,A 87.6435,B 24.8325,C -2.9849,E1 24.987,E2 -4.3987} C_DIS
LIN {X -1.9657,Y 42.8794,Z 66,A 84.6664,B 24.8327,C -2.9835,E1 24.9953,E2 -1.4172} C_DIS
LIN {X 0.5362,Y 42.9214,Z 66,A 81.498,B 24.8324,C -2.9866,E1 25.0042,E2 1.7438} C_DIS
LIN {X 2.6346,Y 42.8441,Z 66,A 78.6689,B 24.8324,C -2.9863,E1 25.0121,E2 4.5726} C_DIS
LIN {X 4.727,Y 42.6633,Z 66,A 75.9126,B 24.8324,C -2.9867,E1 25.0197,E2 7.3263} C_DIS
LIN {X 6.8231,Y 42.3794,Z 66,A 72.9602,B 24.8326,C -2.984,E1 25.0279,E2 10.2822} C_DIS
LIN {X 8.8972,Y 41.9923,Z 66,A 70.2608,B 24.8326,C -2.9845,E1 25.0353,E2 12.9771} C_DIS
LIN {X 11.0606,Y 41.4751,Z 66,A 67.2887,B 24.8328,C -2.9828,E1 25.0433,E2 15.949} C_DIS
LIN {X 13.3497,Y 40.7958,Z 66,A 63.963,B 24.8333,C -2.9783,E1 25.0522,E2 19.2792} C_DIS
LIN {X 15.9997,Y 39.8314,Z 66,A 60.2113,B 24.8337,C -2.975,E1 25.062,E2 23.0307} C_DIS
LIN {X 18.3625,Y 38.7986,Z 66,A 56.9258,B 24.8338,C -2.9736,E1 25.0703,E2 26.3114} C_DIS
LIN {X 20.3449,Y 37.7969,Z 66,A 53.9611,B 24.8342,C -2.9698,E1 25.0777,E2 29.2767} C_DIS
LIN {X 22.4121,Y 36.609,Z 66,A 50.7208,B 24.8349,C -2.9644,E1 25.0855,E2 32.5201} C_DIS
LIN {X 24.3198,Y 35.3709,Z 66,A 47.768,B 24.8352,C -2.9609,E1 25.0923,E2 35.4713} C_DIS
LIN {X 26.218,Y 33.9871,Z 66,A 44.537,B 24.836,C -2.954,E1 25.0995,E2 38.707} C_DIS
LIN {X 28.0905,Y 32.4571,Z 66,A 41.2832,B 24.8367,C -2.9475,E1 25.1065,E2 41.9636} C_DIS
LIN {X 29.8308,Y 30.8647,Z 66,A 38.1893,B 24.8373,C -2.9421,E1 25.1128,E2 45.0576} C_DIS
LIN {X 31.5795,Y 29.0731,Z 66,A 34.9164,B 24.838,C -2.9361,E1 25.1191,E2 48.3306} C_DIS
LIN {X 33.1441,Y 27.2766,Z 66,A 31.7791,B 24.8387,C -2.9296,E1 25.1248,E2 51.469} C_DIS
LIN {X 34.5549,Y 25.4654,Z 66,A 28.7527,B 24.8395,C -2.923,E1 25.1299,E2 54.4967} C_DIS
LIN {X 35.9149,Y 23.5084,Z 66,A 25.5286,B 24.8404,C -2.9143,E1 25.1349,E2 57.7253} C_DIS
LIN {X 37.0827,Y 21.6203,Z 66,A 22.6432,B 24.8411,C -2.908,E1 25.1391,E2 60.611} C_DIS
LIN {X 38.1558,Y 19.6637,Z 66,A 19.6765,B 24.8419,C -2.9002,E1 25.143,E2 63.5804} C_DIS
LIN {X 39.1946,Y 17.5009,Z 66,A 16.3536,B 24.8431,C -2.8894,E1 25.1469,E2 66.9111} C_DIS
LIN {X 40.1926,Y 15.0689,Z 66,A 12.9283,B 24.8441,C -2.8808,E1 25.1504,E2 70.3377} C_DIS
LIN {X 40.9552,Y 12.852,Z 66,A 9.9044,B 24.8449,C -2.8735,E1 25.153,E2 73.3618} C_DIS
LIN {X 41.5743,Y 10.681,Z 66,A 6.808,B 24.846,C -2.8631,E1 25.1553,E2 76.4649} C_DIS
LIN {X 42.1031,Y 8.3583,Z 66,A 3.6768,B 24.8469,C -2.8543,E1 25.1571,E2 79.5987} C_DIS
LIN {X 42.4782,Y 6.1742,Z 66,A 0.8214,B 24.8477,C -2.847,E1 25.1584,E2 82.4546} C_DIS
LIN {X 42.729,Y 4.0934,Z 66,A -1.9883,B 24.8487,C -2.8382,E1 25.1592,E2 85.2686} C_DIS
LIN {X 42.8794,Y 1.9654,Z 66,A -4.9614,B 24.8499,C -2.8271,E1 25.1597,E2 88.2504} C_DIS
LIN {X 42.9195,Y -0.6567,Z 66,A -8.4472,B 24.851,C -2.8163,E1 25.1597,E2 91.7408} C_DIS
LIN {X 42.8087,Y -3.1577,Z 66,A -11.6032,B 24.8518,C -2.8091,E1 25.1592,E2 94.8953} C_DIS
LIN {X 42.5879,Y -5.3663,Z 66,A -14.5206,B 24.8527,C -2.8006,E1 25.1583,E2 97.8155} C_DIS
LIN {X 42.2917,Y -7.3454,Z 66,A -17.1873,B 24.8535,C -2.7923,E1 25.1571,E2 100.4862} C_DIS
LIN {X 41.8542,Y -9.5252,Z 66,A -20.0457,B 24.8543,C -2.7849,E1 25.1554,E2 103.3453} C_DIS
LIN {X 41.3421,Y -11.5473,Z 66,A -22.8691,B 24.8553,C -2.7757,E1 25.1534,E2 106.1744} C_DIS
LIN {X 40.7033,Y -13.6291,Z 66,A -25.7633,B 24.8562,C -2.767,E1 25.1509,E2 109.0727} C_DIS
LIN {X 39.8915,Y -15.8486,Z 66,A -28.9783,B 24.8573,C -2.7564,E1 25.1477,E2 112.2948} C_DIS
LIN {X 38.9728,Y -17.9895,Z 66,A -32.0161,B 24.8581,C -2.7485,E1 25.1443,E2 115.3348} C_DIS
LIN {X 38.0501,Y -19.8667,Z 66,A -34.6448,B 24.8587,C -2.7432,E1 25.141,E2 117.962} C_DIS
LIN {X 37.0993,Y -21.5915,Z 66,A -37.5595,B 24.8599,C -2.7308,E1 25.137,E2 120.891} C_DIS
LIN {X 35.9147,Y -23.5087,Z 66,A -40.5569,B 24.8608,C -2.7226,E1 25.1324,E2 123.8926} C_DIS
LIN {X 34.4825,Y -25.5637,Z 66,A -43.7433,B 24.8614,C -2.7164,E1 25.1273,E2 127.0784} C_DIS
LIN {X 33.001,Y -27.4489,Z 66,A -46.9801,B 24.8623,C -2.7075,E1 25.1216,E2 130.3211} C_DIS
LIN {X 31.4022,Y -29.2651,Z 66,A -50.2707,B 24.8633,C -2.6984,E1 25.1154,E2 133.6185} C_DIS
LIN {X 29.6003,Y -31.0863,Z 66,A -53.5257,B 24.8638,C -2.6931,E1 25.1089,E2 136.8725} C_DIS
LIN {X 27.8467,Y -32.666,Z 66,A -56.7429,B 24.8646,C -2.685,E1 25.1021,E2 140.0963} C_DIS
LIN {X 25.8852,Y -34.2415,Z 66,A -59.6277,B 24.8646,C -2.6857,E1 25.0958,E2 142.9686} C_DIS
LIN {X 23.7884,Y -35.7303,Z 66,A -63.4658,B 24.8659,C -2.6722,E1 25.087,E2 146.8255} C_DIS
LIN {X 21.9315,Y -36.8988,Z 66,A -66.296,B 24.8663,C -2.6685,E1 25.0803,E2 149.6557} C_DIS
LIN {X 20.2183,Y -37.8653,Z 66,A -68.9334,B 24.8668,C -2.6638,E1 25.0738,E2 152.2966} C_DIS
LIN {X 18.2249,Y -38.8635,Z 66,A -71.8668,B 24.8672,C -2.6598,E1 25.0664,E2 155.2318} C_DIS
LIN {X 16.3257,Y -39.6986,Z 66,A -74.5879,B 24.8675,C -2.6566,E1 25.0594,E2 157.954} C_DIS
LIN {X 14.3384,Y -40.4589,Z 66,A -77.4736,B 24.8679,C -2.6521,E1 25.0519,E2 160.8441} C_DIS
LIN {X 12.0674,Y -41.1934,Z 66,A -80.8048,B 24.8685,C -2.6462,E1 25.0429,E2 164.1834} C_DIS
LIN {X 9.8885,Y -41.77,Z 66,A -83.7281,B 24.8687,C -2.6446,E1 25.035,E2 167.1062} C_DIS
LIN {X 7.7182,Y -42.225,Z 66,A -86.7845,B 24.8691,C -2.6407,E1 25.0266,E2 170.1683} C_DIS
LIN {X 5.1248,Y -42.6175,Z 66,A -90.0979,B 24.8691,C -2.6412,E1 25.0175,E2 173.4776} C_DIS
LIN {X 3.0346,Y -42.8172,Z 66,A -93.0613,B 24.8694,C -2.6374,E1 25.0092,E2 176.4483} C_DIS
LIN {X 0.4915,Y -42.9221,Z 66,A -96.3939,B 24.8694,C -2.6374,E1 24.9999,E2 179.7805} C_DIS
LIN {X 0.4915,Y -42.9221,Z 66,A -96.3939,B 24.8694,C -2.6374,E1 24.9999,E2 179.7805} C_DIS
Enddeposition()
LIN {X 0.2039,Y -45.0345,Z 70.5315,A -96.3944,B 24.8694,C -2.6375,E1 24.9999,E2 179.7805} C_DIS
LIN {X 0.188,Y -51.3737,Z 84.1262,A -96.3625,B 24.8707,C -2.6241,E1 24.9999,E2 179.7805} C_DIS
LIN {X 0.188,Y -51.3737,Z 105.1262,A -96.7143,B 24.8557,C -2.7721,E1 24.9999,E2 179.7805} C_DIS
LIN {X 0.4266,Y -66.0765,Z 105.1262,A -95.3195,B 24.8788,C -2.5413,E1 25.0023,E2 178.9345} C_DIS
LIN {X 0.4266,Y -66.0765,Z 85.1262,A -94.9845,B 24.8919,C -2.4004,E1 25.0023,E2 178.9345} C_DIS
LIN {X 0.3488,Y -59.7377,Z 71.5315,A -95.0137,B 24.8908,C -2.4127,E1 25.0023,E2 178.9345} C_DIS
LIN {X 0.3229,Y -57.6248,Z 67,A -95.025,B 24.8903,C -2.4174,E1 25.0023,E2 178.9345} C_DIS
Startdeposition()
$VEL.CP = VEL_PRINT
LIN {X -1.4143,Y -57.6114,Z 67,A -97.7866,B 24.8923,C -2.3961,E1 24.9944,E2 181.7469} C_DIS
LIN {X -4.2394,Y -57.4726,Z 67,A -100.599,B 24.8923,C -2.396,E1 24.9866,E2 184.5604} C_DIS
LIN {X -7.0544,Y -57.1954,Z 67,A -103.4121,B 24.8923,C -2.3963,E1 24.9788,E2 187.3745} C_DIS
LIN {X -9.8523,Y -56.7803,Z 67,A -106.2265,B 24.8922,C -2.397,E1 24.971,E2 190.1897} C_DIS
LIN {X -12.6265,Y -56.2285,Z 67,A -109.0417,B 24.8921,C -2.3982,E1 24.9633,E2 193.0055} C_DIS
LIN {X -15.3703,Y -55.5412,Z 67,A -111.8578,B 24.8919,C -2.3997,E1 24.9557,E2 195.8222} C_DIS
LIN {X -18.0771,Y -54.7201,Z 67,A -114.675,B 24.8918,C -2.4017,E1 24.9482,E2 198.6396} C_DIS
LIN {X -20.7403,Y -53.7672,Z 67,A -117.4932,B 24.8915,C -2.4041,E1 24.9408,E2 201.458} C_DIS
LIN {X -23.3535,Y -52.6848,Z 67,A -120.3122,B 24.8913,C -2.4069,E1 24.9336,E2 204.2769} C_DIS
LIN {X -25.9105,Y -51.4754,Z 67,A -123.1323,B 24.891,C -2.41,E1 24.9265,E2 207.0968} C_DIS
LIN {X -28.4051,Y -50.142,Z 67,A -125.9532,B 24.8907,C -2.4136,E1 24.9196,E2 209.9173} C_DIS
LIN {X -30.8312,Y -48.6879,Z 67,A -128.775,B 24.8903,C -2.4175,E1 24.9129,E2 212.7386} C_DIS
LIN {X -33.1831,Y -47.1164,Z 67,A -131.5979,B 24.8899,C -2.4218,E1 24.9064,E2 215.5607} C_DIS
LIN {X -35.455,Y -45.4314,Z 67,A -134.4213,B 24.8895,C -2.4265,E1 24.9001,E2 218.3833} C_DIS
LIN {X -37.6415,Y -43.637,Z 67,A -137.2441,B 24.889,C -2.4315,E1 24.8941,E2 221.2049} C_DIS
LIN {X -39.7374,Y -41.7375,Z 67,A -140.0709,B 24.8886,C -2.4368,E1 24.8883,E2 224.0305} C_DIS
LIN {X -41.7375,Y -39.7374,Z 67,A -142.8969,B 24.888,C -2.4425,E1 24.8828,E2 226.8551} C_DIS
LIN {X -43.637,Y -37.6415,Z 67,A -145.7236,B 24.8875,C -2.4484,E1 24.8776,E2 229.6803} C_DIS
LIN {X -45.4314,Y -35.455,Z 67,A -148.551,B 24.8869,C -2.4547,E1 24.8727,E2 232.5059} C_DIS
LIN {X -47.1164,Y -33.1831,Z 67,A -151.379,B 24.8863,C -2.4613,E1 24.868,E2 235.3321} C_DIS
LIN {X -48.6879,Y -30.8312,Z 67,A -154.2077,B 24.8857,C -2.4681,E1 24.8637,E2 238.1587} C_DIS
LIN {X -50.142,Y -28.4051,Z 67,A -157.0369,B 24.885,C -2.4751,E1 24.8597,E2 240.9858} C_DIS
LIN {X -51.4754,Y -25.9105,Z 67,A -159.8667,B 24.8843,C -2.4824,E1 24.8561,E2 243.8133} C_DIS
LIN {X -52.6848,Y -23.3535,Z 67,A -162.697,B 24.8836,C -2.4899,E1 24.8528,E2 246.6412} C_DIS
LIN {X -53.7636,Y -20.7494,Z 67,A -165.5204,B 24.8829,C -2.4975,E1 24.8499,E2 249.4621} C_DIS
LIN {X -54.7201,Y -18.0771,Z 67,A -168.3591,B 24.8822,C -2.5054,E1 24.8473,E2 252.298} C_DIS
LIN {X -55.5412,Y -15.3703,Z 67,A -171.1905,B 24.8814,C -2.5135,E1 24.8451,E2 255.1267} C_DIS
LIN {X -56.2285,Y -12.6265,Z 67,A -174.0225,B 24.8806,C -2.5216,E1 24.8433,E2 257.9558} C_DIS
LIN {X -56.7803,Y -9.8523,Z 67,A -176.8546,B 24.8799,C -2.5299,E1 24.8418,E2 260.7849} C_DIS
LIN {X -57.1954,Y -7.0544,Z 67,A -179.687,B 24.8791,C -2.5382,E1 24.8408,E2 263.6142} C_DIS
LIN {X -57.4726,Y -4.2394,Z 67,A 177.4805,B 24.8783,C -2.5467,E1 24.8401,E2 266.4436} C_DIS
LIN {X -57.6114,Y -1.4143,Z 67,A 174.7707,B 24.8772,C -2.5572,E1 24.8398,E2 269.1446} C_DIS
LIN {X -57.6114,Y 1.4143,Z 67,A 171.8151,B 24.8766,C -2.5637,E1 24.8398,E2 272.1024} C_DIS
LIN {X -57.4726,Y 4.2394,Z 67,A 168.9822,B 24.8758,C -2.5722,E1 24.8404,E2 274.9319} C_DIS
LIN {X -57.1954,Y 7.0544,Z 67,A 166.1495,B 24.875,C -2.5807,E1 24.8412,E2 277.7612} C_DIS
LIN {X -56.7803,Y 9.8523,Z 67,A 163.3167,B 24.8741,C -2.5892,E1 24.8425,E2 280.5905} C_DIS
LIN {X -56.2347,Y 12.5982,Z 67,A 160.5059,B 24.8733,C -2.5975,E1 24.8441,E2 283.3982} C_DIS
LIN {X -55.5412,Y 15.3703,Z 67,A 157.6518,B 24.8725,C -2.6061,E1 24.8461,E2 286.2485} C_DIS
LIN {X -54.7201,Y 18.0771,Z 67,A 154.8197,B 24.8717,C -2.6143,E1 24.8485,E2 289.077} C_DIS
LIN {X -53.7672,Y 20.7403,Z 67,A 151.9877,B 24.8709,C -2.6225,E1 24.8513,E2 291.9055} C_DIS
LIN {X -52.6848,Y 23.3535,Z 67,A 149.1562,B 24.8701,C -2.6305,E1 24.8544,E2 294.7334} C_DIS
LIN {X -51.4754,Y 25.9105,Z 67,A 146.3248,B 24.8693,C -2.6384,E1 24.8578,E2 297.5612} C_DIS
LIN {X -50.142,Y 28.4051,Z 67,A 143.494,B 24.8685,C -2.6462,E1 24.8616,E2 300.3885} C_DIS
LIN {X -48.6879,Y 30.8312,Z 67,A 140.6637,B 24.8678,C -2.6537,E1 24.8658,E2 303.2153} C_DIS
LIN {X -47.1164,Y 33.1831,Z 67,A 137.8336,B 24.867,C -2.661,E1 24.8702,E2 306.0419} C_DIS
LIN {X -45.4314,Y 35.455,Z 67,A 135.0042,B 24.8663,C -2.6681,E1 24.875,E2 308.8678} C_DIS
LIN {X -43.637,Y 37.6415,Z 67,A 132.1755,B 24.8656,C -2.6749,E1 24.8801,E2 311.6932} C_DIS
LIN {X -41.7375,Y 39.7374,Z 67,A 129.3474,B 24.865,C -2.6815,E1 24.8855,E2 314.518} C_DIS
LIN {X -39.7374,Y 41.7375,Z 67,A 126.5198,B 24.8643,C -2.6879,E1 24.8911,E2 317.3423} C_DIS
LIN {X -37.6415,Y 43.637,Z 67,A 123.693,B 24.8637,C -2.6939,E1 24.897,E2 320.1659} C_DIS
LIN {X -35.455,Y 45.4314,Z 67,A 120.8669,B 24.8631,C -2.6996,E1 24.9032,E2 322.9889} C_DIS
LIN {X -33.1831,Y 47.1164,Z 67,A 118.0415,B 24.8626,C -2.705,E1 24.9095,E2 325.8112} C_DIS
LIN {X -30.8312,Y 48.6879,Z 67,A 115.217,B 24.8621,C -2.7101,E1 24.9161,E2 328.6329} C_DIS
LIN {X -28.4051,Y 50.142,Z 67,A 112.3933,B 24.8616,C -2.7148,E1 24.9229,E2 331.4538} C_DIS
LIN {X -25.9105,Y 51.4754,Z 67,A 109.5703,B 24.8611,C -2.7192,E1 24.9299,E2 334.274} C_DIS
LIN {X -23.3535,Y 52.6848,Z 67,A 106.7483,B 24.8607,C -2.7232,E1 24.9371,E2 337.0935} C_DIS
LIN {X -20.7403,Y 53.7672,Z 67,A 103.9271,B 24.8604,C -2.7268,E1 24.9444,E2 339.9122} C_DIS
LIN {X -18.0771,Y 54.7201,Z 67,A 101.1068,B 24.86,C -2.7301,E1 24.9518,E2 342.7301} C_DIS
LIN {X -15.3703,Y 55.5412,Z 67,A 98.2876,B 24.8597,C -2.7329,E1 24.9594,E2 345.5471} C_DIS
LIN {X -12.6265,Y 56.2285,Z 67,A 95.4691,B 24.8595,C -2.7354,E1 24.967,E2 348.3636} C_DIS
LIN {X -9.8523,Y 56.7803,Z 67,A 92.6518,B 24.8593,C -2.7375,E1 24.9748,E2 351.179} C_DIS
LIN {X -7.0544,Y 57.1954,Z 67,A 89.8353,B 24.8591,C -2.7391,E1 24.9826,E2 353.9937} C_DIS
LIN {X -4.2394,Y 57.4726,Z 67,A 87.0199,B 24.859,C -2.7404,E1 24.9904,E2 356.8075} C_DIS
LIN {X -1.4143,Y 57.6114,Z 67,A 84.2054,B 24.8589,C -2.7412,E1 24.9982,E2 359.6204} C_DIS
LIN {X 1.4143,Y 57.6114,Z 67,A 81.3919,B 24.8589,C -2.7416,E1 25.0061,E2 362.4326} C_DIS
LIN {X 4.2394,Y 57.4726,Z 67,A 78.5793,B 24.8589,C -2.7416,E1 25.0139,E2 365.2441} C_DIS
LIN {X 7.0544,Y 57.1954,Z 67,A 75.7679,B 24.8589,C -2.7412,E1 25.0217,E2 368.0546} C_DIS
LIN {X 9.8523,Y 56.7803,Z 67,A 72.9573,B 24.8589,C -2.7404,E1 25.0295,E2 370.8644} C_DIS
LIN {X 12.6265,Y 56.2285,Z 67,A 70.1478,B 24.8591,C -2.7391,E1 25.0371,E2 373.6732} C_DIS
LIN {X 15.3703,Y 55.5412,Z 67,A 67.3393,B 24.8593,C -2.7375,E1 25.0447,E2 376.4813} C_DIS
LIN {X 18.0771,Y 54.7201,Z 67,A 64.5408,B 24.8594,C -2.7356,E1 25.0522,E2 379.2791} C_DIS
LIN {X 20.7403,Y 53.7672,Z 67,A 61.7249,B 24.8597,C -2.733,E1 25.0596,E2 382.0953} C_DIS
LIN {X 23.3536,Y 52.6848,Z 67,A 58.9193,B 24.86,C -2.7301,E1 25.0668,E2 384.9009} C_DIS
LIN {X 25.9105,Y 51.4754,Z 67,A 56.1144,B 24.8603,C -2.7269,E1 25.0738,E2 387.7061} C_DIS
LIN {X 28.3616,Y 50.1663,Z 67,A 53.3469,B 24.8607,C -2.7231,E1 25.0806,E2 390.4746} C_DIS
LIN {X 30.8312,Y 48.6879,Z 67,A 50.5075,B 24.8611,C -2.7193,E1 25.0873,E2 393.3139} C_DIS
LIN {X 33.1831,Y 47.1164,Z 67,A 47.7052,B 24.8616,C -2.715,E1 25.0938,E2 396.1169} C_DIS
LIN {X 35.455,Y 45.4314,Z 67,A 44.904,B 24.862,C -2.7103,E1 25.1,E2 398.9191} C_DIS
LIN {X 37.6415,Y 43.637,Z 67,A 42.1035,B 24.8626,C -2.7053,E1 25.106,E2 401.7207} C_DIS
LIN {X 39.7374,Y 41.7375,Z 67,A 39.3036,B 24.8631,C -2.6999,E1 25.1117,E2 404.5218} C_DIS
LIN {X 41.7375,Y 39.7374,Z 67,A 36.5045,B 24.8637,C -2.6943,E1 25.1172,E2 407.3223} C_DIS
LIN {X 43.637,Y 37.6415,Z 67,A 33.7061,B 24.8643,C -2.6883,E1 25.1224,E2 410.1223} C_DIS
LIN {X 45.4314,Y 35.455,Z 67,A 30.9085,B 24.8649,C -2.6821,E1 25.1273,E2 412.9216} C_DIS
LIN {X 47.1164,Y 33.1831,Z 67,A 28.1116,B 24.8656,C -2.6756,E1 25.1318,E2 415.7204} C_DIS
LIN {X 48.6879,Y 30.8312,Z 67,A 25.3151,B 24.8662,C -2.6688,E1 25.1361,E2 418.5189} C_DIS
LIN {X 50.142,Y 28.4051,Z 67,A 22.5193,B 24.867,C -2.6618,E1 25.14,E2 421.3169} C_DIS
LIN {X 51.4754,Y 25.9105,Z 67,A 19.7239,B 24.8677,C -2.6546,E1 25.1436,E2 424.1145} C_DIS
LIN {X 52.6848,Y 23.3535,Z 67,A 16.9292,B 24.8684,C -2.6472,E1 25.1469,E2 426.9116} C_DIS
LIN {X 53.7672,Y 20.7403,Z 67,A 14.1346,B 24.8692,C -2.6396,E1 25.1498,E2 429.7087} C_DIS
LIN {X 54.7201,Y 18.0771,Z 67,A 11.3406,B 24.8699,C -2.6318,E1 25.1523,E2 432.5055} C_DIS
LIN {X 55.5412,Y 15.3703,Z 67,A 8.547,B 24.8707,C -2.6239,E1 25.1545,E2 435.3019} C_DIS
LIN {X 56.2285,Y 12.6265,Z 67,A 5.7537,B 24.8715,C -2.6158,E1 25.1563,E2 438.098} C_DIS
LIN {X 56.7803,Y 9.8523,Z 67,A 2.9605,B 24.8723,C -2.6076,E1 25.1577,E2 440.8941} C_DIS
LIN {X 57.1954,Y 7.0544,Z 67,A 0.1677,B 24.8731,C -2.5994,E1 25.1588,E2 443.6901} C_DIS
LIN {X 57.4726,Y 4.2394,Z 67,A -2.625,B 24.874,C -2.591,E1 25.1595,E2 446.4859} C_DIS
LIN {X 57.6114,Y 1.4143,Z 67,A -5.2965,B 24.8745,C -2.5854,E1 25.1598,E2 449.1548} C_DIS
LIN {X 57.6244,Y -0.7072,Z 67,A -7.1785,B 24.8746,C -2.584,E1 25.1598,E2 451.0288} C_DIS
LIN {X 57.5593,Y -2.8277,Z 67,A -9.6062,B 24.876,C -2.57,E1 25.1595,E2 453.4752} C_DIS
LIN {X 57.3512,Y -5.6486,Z 67,A -12.3986,B 24.8768,C -2.5616,E1 25.1588,E2 456.2711} C_DIS
LIN {X 57.005,Y -8.4559,Z 67,A -15.1912,B 24.8776,C -2.5532,E1 25.1578,E2 459.067} C_DIS
LIN {X 56.5214,Y -11.2428,Z 67,A -17.9836,B 24.8784,C -2.5448,E1 25.1563,E2 461.863} C_DIS
LIN {X 55.9017,Y -14.0026,Z 67,A -20.7765,B 24.8792,C -2.5365,E1 25.1545,E2 464.6593} C_DIS
LIN {X 55.1473,Y -16.7287,Z 67,A -23.5693,B 24.88,C -2.5282,E1 25.1524,E2 467.4556} C_DIS
LIN {X 54.26,Y -19.4145,Z 67,A -26.3625,B 24.8808,C -2.5201,E1 25.1498,E2 470.2524} C_DIS
LIN {X 53.2563,Y -22.0184,Z 67,A -29.1281,B 24.8816,C -2.5119,E1 25.147,E2 473.0219} C_DIS
LIN {X 52.0958,Y -24.6395,Z 67,A -31.9496,B 24.8823,C -2.5041,E1 25.1437,E2 475.8465} C_DIS
LIN {X 50.824,Y -27.166,Z 67,A -34.7437,B 24.883,C -2.4964,E1 25.1401,E2 478.6442} C_DIS
LIN {X 49.4298,Y -29.6271,Z 67,A -37.5265,B 24.8837,C -2.4891,E1 25.1362,E2 481.4299} C_DIS
LIN {X 47.9166,Y -32.0168,Z 67,A -40.3331,B 24.8844,C -2.4814,E1 25.1319,E2 484.2406} C_DIS
LIN {X 46.2878,Y -34.3294,Z 67,A -43.1286,B 24.8851,C -2.4742,E1 25.1273,E2 487.0395} C_DIS
LIN {X 44.5476,Y -36.5593,Z 67,A -45.9245,B 24.8857,C -2.4673,E1 25.1224,E2 489.8388} C_DIS
LIN {X 42.7001,Y -38.7011,Z 67,A -48.7211,B 24.8864,C -2.4606,E1 25.1173,E2 492.6387} C_DIS
LIN {X 40.7497,Y -40.7497,Z 67,A -51.5183,B 24.887,C -2.4541,E1 25.1118,E2 495.4392} C_DIS
LIN {X 38.7011,Y -42.7001,Z 67,A -54.316,B 24.8875,C -2.4479,E1 25.1061,E2 498.2402} C_DIS
LIN {X 36.5593,Y -44.5476,Z 67,A -57.1145,B 24.8881,C -2.442,E1 25.1001,E2 501.0419} C_DIS
LIN {X 34.3294,Y -46.2878,Z 67,A -59.9137,B 24.8886,C -2.4364,E1 25.0939,E2 503.844} C_DIS
LIN {X 32.0168,Y -47.9166,Z 67,A -62.7137,B 24.8891,C -2.4312,E1 25.0874,E2 506.6471} C_DIS
LIN {X 29.6271,Y -49.4298,Z 67,A -65.5145,B 24.8895,C -2.4262,E1 25.0807,E2 509.4507} C_DIS
LIN {X 27.166,Y -50.824,Z 67,A -68.3159,B 24.8899,C -2.4216,E1 25.0739,E2 512.2549} C_DIS
LIN {X 24.6395,Y -52.0958,Z 67,A -71.1185,B 24.8903,C -2.4173,E1 25.0669,E2 515.0601} C_DIS
LIN {X 22.0536,Y -53.242,Z 67,A -73.9215,B 24.8907,C -2.4134,E1 25.0597,E2 517.8657} C_DIS
LIN {X 19.4145,Y -54.26,Z 67,A -76.7258,B 24.891,C -2.4099,E1 25.0523,E2 520.6724} C_DIS
LIN {X 16.7287,Y -55.1473,Z 67,A -79.5308,B 24.8913,C -2.4068,E1 25.0448,E2 523.4797} C_DIS
LIN {X 14.0026,Y -55.9017,Z 67,A -82.3367,B 24.8915,C -2.404,E1 25.0373,E2 526.2877} C_DIS
LIN {X 11.2428,Y -56.5214,Z 67,A -85.1435,B 24.8918,C -2.4017,E1 25.0296,E2 529.0966} C_DIS
LIN {X 8.4559,Y -57.005,Z 67,A -87.9515,B 24.8919,C -2.3997,E1 25.0218,E2 531.9064} C_DIS
LIN {X 5.6486,Y -57.3512,Z 67,A -90.7602,B 24.8921,C -2.3982,E1 25.014,E2 534.7168} C_DIS
LIN {X 2.8277,Y -57.5593,Z 67,A -93.5701,B 24.8921,C -2.397,E1 25.0062,E2 537.5283} C_DIS
LIN {X 0.3229,Y -57.6248,Z 67,A -95.0247,B 24.8903,C -2.4174,E1 25.0023,E2 538.9342} C_DIS
Enddeposition()
LIN {X 0.3229,Y -57.6248,Z 67,A -95.0247,B 24.8903,C -2.4174,E1 25.0023,E2 538.9342} C_DIS
Startdeposition()
$VEL.CP = VEL_PRINT
LIN {X 1.8385,Y -56.6104,Z 67,A -93.1944,B 24.8882,C -2.4408,E1 25.0076,E2 537.0486} C_DIS
LIN {X 4.7135,Y -56.4441,Z 67,A -90.3355,B 24.8882,C -2.441,E1 25.0155,E2 534.1905} C_DIS
LIN {X 8.1714,Y -56.048,Z 67,A -86.7704,B 24.8879,C -2.4442,E1 25.0254,E2 530.6209} C_DIS
LIN {X 9.9677,Y -55.7562,Z 67,A -84.4302,B 24.8868,C -2.456,E1 25.0319,E2 528.2551} C_DIS
LIN {X 13.576,Y -54.9893,Z 67,A -81.2492,B 24.8875,C -2.4479,E1 25.0405,E2 525.0977} C_DIS
LIN {X 16.2001,Y -54.2741,Z 67,A -78.5463,B 24.8874,C -2.4499,E1 25.0477,E2 522.3947} C_DIS
LIN {X 18.6234,Y -53.4911,Z 67,A -76.1972,B 24.8875,C -2.4482,E1 25.0539,E2 520.0541} C_DIS
LIN {X 21.0563,Y -52.5818,Z 67,A -73.3275,B 24.8867,C -2.4569,E1 25.0615,E2 517.1701} C_DIS
LIN {X 23.3673,Y -51.5954,Z 67,A -70.8117,B 24.8864,C -2.4601,E1 25.0679,E2 514.6527} C_DIS
LIN {X 25.8438,Y -50.4005,Z 67,A -67.8567,B 24.8856,C -2.4683,E1 25.0753,E2 511.6862} C_DIS
LIN {X 28.5693,Y -48.908,Z 67,A -64.6988,B 24.8851,C -2.4742,E1 25.083,E2 508.524} C_DIS
LIN {X 31.7535,Y -46.9023,Z 67,A -61.4794,B 24.8856,C -2.4686,E1 25.0905,E2 505.3283} C_DIS
LIN {X 34.024,Y -45.2821,Z 67,A -58.1405,B 24.884,C -2.4857,E1 25.0981,E2 501.9607} C_DIS
LIN {X 36.4713,Y -43.3368,Z 67,A -55.0842,B 24.8836,C -2.4902,E1 25.1047,E2 498.9054} C_DIS
LIN {X 38.5933,Y -41.4578,Z 67,A -52.2582,B 24.8831,C -2.4958,E1 25.1105,E2 496.0774} C_DIS
LIN {X 40.4252,Y -39.673,Z 67,A -49.4522,B 24.882,C -2.5069,E1 25.1161,E2 493.257} C_DIS
LIN {X 42.8601,Y -37.0299,Z 67,A -46.2149,B 24.882,C -2.507,E1 25.1221,E2 490.0338} C_DIS
LIN {X 44.8175,Y -34.6339,Z 67,A -42.3984,B 24.8798,C -2.5308,E1 25.1288,E2 486.179} C_DIS
LIN {X 46.5446,Y -32.2756,Z 67,A -39.3023,B 24.8787,C -2.542,E1 25.1337,E2 483.0715} C_DIS
LIN {X 48.8603,Y -28.6499,Z 67,A -35.6599,B 24.8791,C -2.5379,E1 25.139,E2 479.4573} C_DIS
LIN {X 50.2365,Y -26.1624,Z 67,A -32.9056,B 24.8786,C -2.5434,E1 25.1426,E2 476.7045} C_DIS
LIN {X 51.1757,Y -24.2735,Z 67,A -30.316,B 24.8769,C -2.5602,E1 25.1458,E2 474.0892} C_DIS
LIN {X 52.6214,Y -20.9565,Z 67,A -27.08,B 24.8769,C -2.5614,E1 25.1492,E2 470.8683} C_DIS
LIN {X 53.5951,Y -18.3229,Z 67,A -24.3394,B 24.8762,C -2.5677,E1 25.1518,E2 468.128} C_DIS
LIN {X 54.335,Y -15.9946,Z 67,A -21.8318,B 24.8754,C -2.5762,E1 25.1538,E2 465.6147} C_DIS
LIN {X 55.2199,Y -12.6052,Z 67,A -18.2635,B 24.8743,C -2.5878,E1 25.1562,E2 462.0396} C_DIS
LIN {X 55.6882,Y -10.3452,Z 67,A -15.6996,B 24.873,C -2.6004,E1 25.1576,E2 459.4609} C_DIS
LIN {X 56.2121,Y -6.9576,Z 67,A -12.4836,B 24.8725,C -2.6055,E1 25.1588,E2 456.2518} C_DIS
LIN {X 56.4965,Y -4.0376,Z 67,A -9.518,B 24.8716,C -2.6148,E1 25.1595,E2 453.2817} C_DIS
LIN {X 56.6043,Y -2.0375,Z 67,A -7.6026,B 24.8712,C -2.6187,E1 25.1597,E2 451.3686} C_DIS
LIN {X 56.6371,Y 0.6775,Z 67,A -4.8769,B 24.8704,C -2.6268,E1 25.1597,E2 448.6398} C_DIS
LIN {X 56.5359,Y 3.4501,Z 67,A -2.0565,B 24.8695,C -2.636,E1 25.1593,E2 445.8146} C_DIS
LIN {X 56.285,Y 6.338,Z 67,A 0.5271,B 24.8695,C -2.6371,E1 25.1587,E2 443.2436} C_DIS
LIN {X 56.072,Y 8.0024,Z 67,A 2.5702,B 24.8681,C -2.6503,E1 25.1579,E2 441.1813} C_DIS
LIN {X 55.5756,Y 10.932,Z 67,A 5.5201,B 24.8673,C -2.6582,E1 25.1564,E2 438.23} C_DIS
LIN {X 54.9564,Y 13.711,Z 67,A 8.4386,B 24.8664,C -2.6678,E1 25.1545,E2 435.3058} C_DIS
LIN {X 53.7898,Y 17.7447,Z 67,A 12.6834,B 24.8651,C -2.6802,E1 25.1511,E2 431.0557} C_DIS
LIN {X 52.8083,Y 20.4804,Z 67,A 15.7605,B 24.8639,C -2.6918,E1 25.148,E2 427.9684} C_DIS
LIN {X 51.5124,Y 23.5517,Z 67,A 18.7792,B 24.8638,C -2.6932,E1 25.1447,E2 424.9628} C_DIS
LIN {X 50.3969,Y 25.8509,Z 67,A 21.4159,B 24.8629,C -2.7015,E1 25.1414,E2 422.3206} C_DIS
LIN {X 49.2252,Y 28.0186,Z 67,A 23.8193,B 24.8625,C -2.7061,E1 25.1381,E2 419.9189} C_DIS
LIN {X 48.344,Y 29.5123,Z 67,A 25.5023,B 24.8622,C -2.709,E1 25.1357,E2 418.2374} C_DIS
LIN {X 46.4834,Y 32.3636,Z 67,A 29.6891,B 24.8596,C -2.7343,E1 25.1291,E2 414.0117} C_DIS
LIN {X 44.0658,Y 35.5855,Z 67,A 33.5933,B 24.859,C -2.74,E1 25.1224,E2 410.1122} C_DIS
LIN {X 41.5497,Y 38.4943,Z 67,A 37.039,B 24.8591,C -2.7388,E1 25.116,E2 406.6848} C_DIS
LIN {X 39.5226,Y 40.573,Z 67,A 39.8881,B 24.8587,C -2.743,E1 25.1103,E2 403.8378} C_DIS
LIN {X 37.8994,Y 42.0924,Z 67,A 41.9044,B 24.8587,C -2.7424,E1 25.1062,E2 401.8311} C_DIS
LIN {X 35.7735,Y 43.913,Z 67,A 45.5254,B 24.8564,C -2.7648,E1 25.0984,E2 398.171} C_DIS
LIN {X 32.0612,Y 46.6934,Z 67,A 49.7276,B 24.8567,C -2.7621,E1 25.0889,E2 393.9898} C_DIS
LIN {X 29.6402,Y 48.2663,Z 67,A 52.5298,B 24.8565,C -2.764,E1 25.0823,E2 391.1921} C_DIS
LIN {X 27.1673,Y 49.6999,Z 67,A 55.3403,B 24.8563,C -2.7663,E1 25.0755,E2 388.3846} C_DIS
LIN {X 25.1522,Y 50.7492,Z 67,A 57.7134,B 24.8558,C -2.7707,E1 25.0695,E2 386.0074} C_DIS
LIN {X 23.2064,Y 51.6679,Z 67,A 59.941,B 24.8554,C -2.7743,E1 25.0639,E2 383.777} C_DIS
LIN {X 20.6395,Y 52.7459,Z 67,A 63.7784,B 24.8529,C -2.7983,E1 25.0538,E2 379.8911} C_DIS
LIN {X 17.3173,Y 53.9281,Z 67,A 65.9067,B 24.8557,C -2.7715,E1 25.0483,E2 377.8306} C_DIS
LIN {X 15.094,Y 54.5927,Z 67,A 68.6704,B 24.8547,C -2.7816,E1 25.0409,E2 375.0477} C_DIS
LIN {X 12.6138,Y 55.2179,Z 67,A 71.2771,B 24.8545,C -2.7833,E1 25.0338,E2 372.4404} C_DIS
LIN {X 10.2926,Y 55.6978,Z 67,A 73.5978,B 24.8545,C -2.7828,E1 25.0274,E2 370.1238} C_DIS
LIN {X 7.4445,Y 56.1491,Z 67,A 76.5372,B 24.8545,C -2.784,E1 25.0193,E2 367.1841} C_DIS
LIN {X 4.6581,Y 56.4485,Z 67,A 79.3023,B 24.8545,C -2.7829,E1 25.0116,E2 364.4234} C_DIS
LIN {X 1.9073,Y 56.6083,Z 67,A 81.9381,B 24.8548,C -2.7798,E1 25.0043,E2 361.7958} C_DIS
LIN {X -0.5185,Y 56.6381,Z 67,A 85.3252,B 24.853,C -2.7975,E1 24.9947,E2 358.3666} C_DIS
LIN {X -4.8173,Y 56.4358,Z 67,A 89.0104,B 24.8545,C -2.7828,E1 24.9846,E2 354.7151} C_DIS
LIN {X -7.752,Y 56.1076,Z 67,A 92.3894,B 24.8539,C -2.7885,E1 24.9752,E2 351.32} C_DIS
LIN {X -11.9076,Y 55.3746,Z 67,A 96.2414,B 24.8551,C -2.7773,E1 24.9647,E2 347.4906} C_DIS
LIN {X -15.1549,Y 54.5746,Z 67,A 99.6965,B 24.8553,C -2.7753,E1 24.9553,E2 344.0351} C_DIS
LIN {X -17.6182,Y 53.8307,Z 67,A 102.219,B 24.8558,C -2.7709,E1 24.9486,E2 341.5187} C_DIS
LIN {X -19.9698,Y 53.0031,Z 67,A 104.8778,B 24.8558,C -2.7702,E1 24.9416,E2 338.8561} C_DIS
LIN {X -22.655,Y 51.912,Z 67,A 107.58,B 24.8567,C -2.7619,E1 24.9347,E2 336.1674} C_DIS
LIN {X -25.0692,Y 50.7903,Z 67,A 110.3218,B 24.8571,C -2.7587,E1 24.9278,E2 333.4264} C_DIS
LIN {X -27.4584,Y 49.5396,Z 67,A 113.0094,B 24.8576,C -2.7534,E1 24.9212,E2 330.7438} C_DIS
LIN {X -29.4226,Y 48.3986,Z 67,A 115.2854,B 24.8581,C -2.749,E1 24.9158,E2 328.4715} C_DIS
LIN {X -31.1476,Y 47.3068,Z 67,A 117.4135,B 24.8584,C -2.7462,E1 24.9108,E2 326.343} C_DIS
LIN {X -33.271,Y 45.8389,Z 67,A 120.1338,B 24.8587,C -2.743,E1 24.9046,E2 323.6211} C_DIS
LIN {X -35.503,Y 44.1327,Z 67,A 122.9797,B 24.8593,C -2.7371,E1 24.8983,E2 320.7788} C_DIS
LIN {X -37.4065,Y 42.5312,Z 67,A 125.4682,B 24.8599,C -2.7311,E1 24.8931,E2 318.2949} C_DIS
LIN {X -39.1398,Y 40.9419,Z 67,A 127.6446,B 24.8608,C -2.7221,E1 24.8886,E2 316.131} C_DIS
LIN {X -40.2773,Y 39.8227,Z 67,A 129.5399,B 24.8608,C -2.7231,E1 24.8849,E2 314.2253} C_DIS
LIN {X -42.0996,Y 37.8914,Z 67,A 132.3168,B 24.8612,C -2.7181,E1 24.8796,E2 311.4481} C_DIS
LIN {X -43.9032,Y 35.786,Z 67,A 135.038,B 24.8621,C -2.7096,E1 24.8748,E2 308.7348} C_DIS
LIN {X -45.3307,Y 33.9594,Z 67,A 137.2354,B 24.863,C -2.7009,E1 24.8711,E2 306.5476} C_DIS
LIN {X -46.5026,Y 32.3361,Z 67,A 139.6005,B 24.863,C -2.7012,E1 24.8672,E2 304.1702} C_DIS
LIN {X -48.0793,Y 29.9415,Z 67,A 142.4283,B 24.8639,C -2.692,E1 24.863,E2 301.3501} C_DIS
LIN {X -49.5685,Y 27.4068,Z 67,A 145.4306,B 24.8647,C -2.684,E1 24.8589,E2 298.3511} C_DIS
LIN {X -50.9323,Y 24.7807,Z 67,A 148.4926,B 24.8655,C -2.6765,E1 24.855,E2 295.2907} C_DIS
LIN {X -52.0473,Y 22.3449,Z 67,A 151.1994,B 24.8663,C -2.6684,E1 24.852,E2 292.5883} C_DIS
LIN {X -52.769,Y 20.5805,Z 67,A 153.323,B 24.8665,C -2.6659,E1 24.8498,E2 290.4588} C_DIS
LIN {X -53.6051,Y 18.2934,Z 67,A 155.465,B 24.8678,C -2.6531,E1 24.8479,E2 288.3354} C_DIS
Enddeposition()
END
